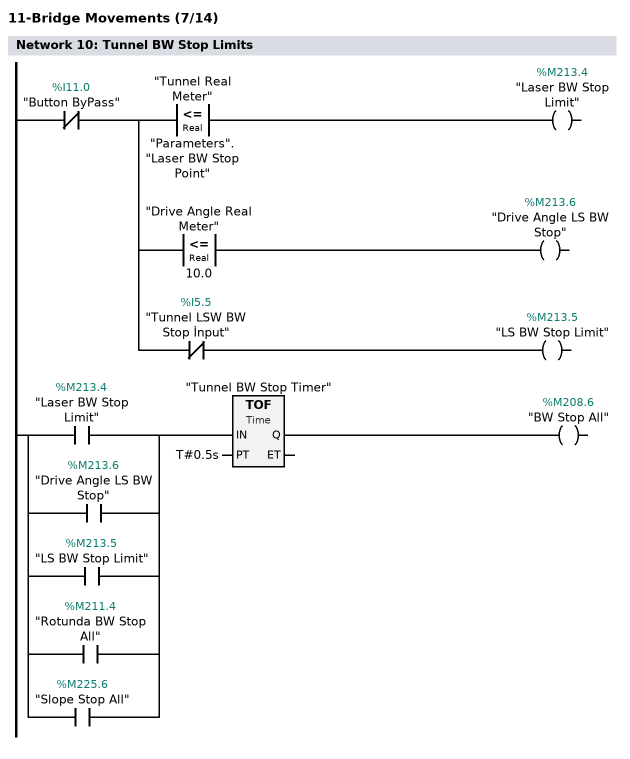
   RUNG wire#powerrail
      I_Contact( "Button ByPass" )
      wire#w1
      { S7_Templates := "SrcType := Real" } LE_Contact(in1 := "Tunnel Real Meter", in2 := "Parameters"."Laser BW Stop Point")
      Coil( "Laser BW Stop Limit" )
   END_RUNG
   RUNG wire#w1
      { S7_Templates := "SrcType := Real" } LE_Contact(in1 := "Drive Angle Real Meter", in2 := 10.0)
      Coil( "Drive Angle LS BW Stop" )
   END_RUNG
   RUNG wire#w1
      I_Contact( "Tunnel LSW BW Stop İnput" )
      Coil( "LS BW Stop Limit" )
   END_RUNG
   RUNG wire#powerrail
      Contact( "Laser BW Stop Limit" )
      wire#w2
      { S7_Templates := "time_type := Time" } "Tunnel BW Stop Timer".TOF(pt := T#0.5s, et =>)
      Coil( "BW Stop All" )
   END_RUNG
   RUNG wire#powerrail
      Contact( "Drive Angle LS BW Stop" )
   END_RUNG wire#w2
   RUNG wire#powerrail
      Contact( "LS BW Stop Limit" )
   END_RUNG wire#w2
   RUNG wire#powerrail
      Contact( "Rotunda BW Stop All" )
   END_RUNG wire#w2
   RUNG wire#powerrail
      Contact( "Slope Stop All" )
   END_RUNG wire#w2
   // the same network as SCL:
   "Laser BW Stop Limit" := NOT "Button ByPass" AND ("Tunnel Real Meter" <= "Parameters"."Laser BW Stop Point");
   "Drive Angle LS BW Stop" := NOT "Button ByPass" AND ("Drive Angle Real Meter" <= 10.0);
   "LS BW Stop Limit" := NOT "Button ByPass" AND NOT "Tunnel LSW BW Stop İnput";
   "Tunnel BW Stop Timer".TOF(IN := "Laser BW Stop Limit" OR "Drive Angle LS BW Stop" OR "LS BW Stop Limit" OR "Rotunda BW Stop All" OR "Slope Stop All",
                           PT := T#0.5s);
   "BW Stop All" := "Tunnel BW Stop Timer".Q;
END_REGION

REGION Network 11: Tunnel FW
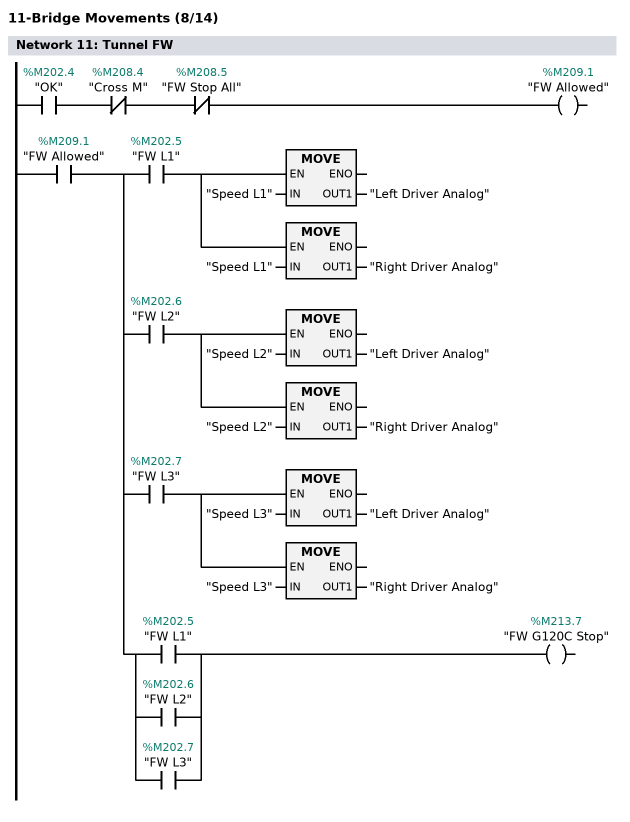
   RUNG wire#powerrail
      Contact( "OK" )
      I_Contact( "Cross M" )
      I_Contact( "FW Stop All" )
      Coil( "FW Allowed" )
   END_RUNG
   RUNG wire#powerrail
      Contact( "FW Allowed" )
      wire#w1
      Contact( "FW L1" )
      wire#w2
      Move(in := "Speed L1", out1 => "Left Driver Analog")
   END_RUNG
   RUNG wire#w2
      Move(in := "Speed L1", out1 => "Right Driver Analog")
   END_RUNG
   RUNG wire#w1
      Contact( "FW L2" )
      wire#w3
      Move(in := "Speed L2", out1 => "Left Driver Analog")
   END_RUNG
   RUNG wire#w3
      Move(in := "Speed L2", out1 => "Right Driver Analog")
   END_RUNG
   RUNG wire#w1
      Contact( "FW L3" )
      wire#w4
      Move(in := "Speed L3", out1 => "Left Driver Analog")
   END_RUNG
   RUNG wire#w4
      Move(in := "Speed L3", out1 => "Right Driver Analog")
   END_RUNG
   RUNG wire#w1
      Contact( "FW L1" )
      wire#w5
      Coil( "FW G120C Stop" )
   END_RUNG
   RUNG wire#w1
      Contact( "FW L2" )
   END_RUNG wire#w5
   RUNG wire#w1
      Contact( "FW L3" )
   END_RUNG wire#w5
   // the same network as SCL:
   "FW Allowed" := "OK" AND NOT "Cross M" AND NOT "FW Stop All";
   IF "FW Allowed" AND "FW L1" THEN
       "Left Driver Analog" := "Speed L1";
       "Right Driver Analog" := "Speed L1";
   END_IF;
   IF "FW Allowed" AND "FW L2" THEN
       "Left Driver Analog" := "Speed L2";
       "Right Driver Analog" := "Speed L2";
   END_IF;
   IF "FW Allowed" AND "FW L3" THEN
       "Left Driver Analog" := "Speed L3";
       "Right Driver Analog" := "Speed L3";
   END_IF;
   "FW G120C Stop" := "FW Allowed" AND ("FW L1" OR "FW L2" OR "FW L3");
END_REGION

REGION Network 12: Tunnel BW
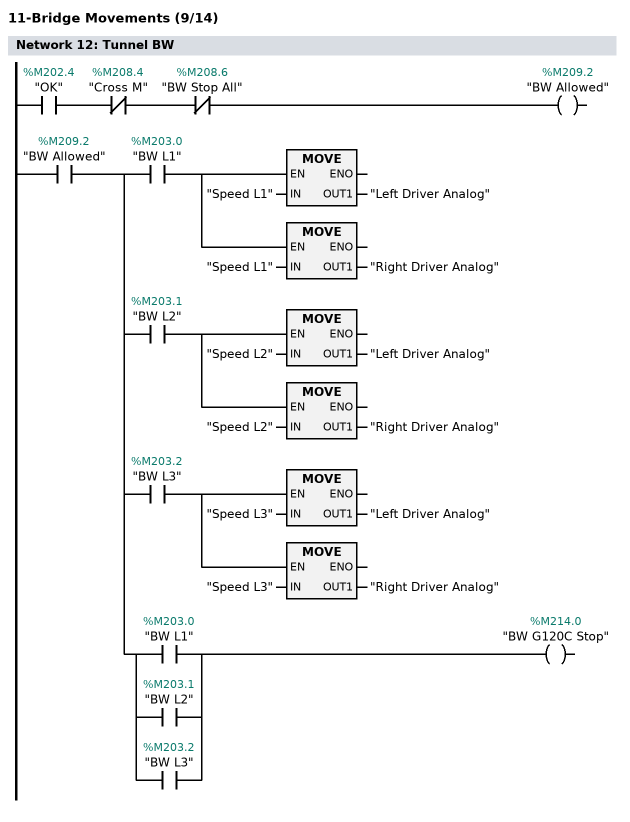
   RUNG wire#powerrail
      Contact( "OK" )
      I_Contact( "Cross M" )
      I_Contact( "BW Stop All" )
      Coil( "BW Allowed" )
   END_RUNG
   RUNG wire#powerrail
      Contact( "BW Allowed" )
      wire#w1
      Contact( "BW L1" )
      wire#w2
      Move(in := "Speed L1", out1 => "Left Driver Analog")
   END_RUNG
   RUNG wire#w2
      Move(in := "Speed L1", out1 => "Right Driver Analog")
   END_RUNG
   RUNG wire#w1
      Contact( "BW L2" )
      wire#w3
      Move(in := "Speed L2", out1 => "Left Driver Analog")
   END_RUNG
   RUNG wire#w3
      Move(in := "Speed L2", out1 => "Right Driver Analog")
   END_RUNG
   RUNG wire#w1
      Contact( "BW L3" )
      wire#w4
      Move(in := "Speed L3", out1 => "Left Driver Analog")
   END_RUNG
   RUNG wire#w4
      Move(in := "Speed L3", out1 => "Right Driver Analog")
   END_RUNG
   RUNG wire#w1
      Contact( "BW L1" )
      wire#w5
      Coil( "BW G120C Stop" )
   END_RUNG
   RUNG wire#w1
      Contact( "BW L2" )
   END_RUNG wire#w5
   RUNG wire#w1
      Contact( "BW L3" )
   END_RUNG wire#w5
   // the same network as SCL:
   "BW Allowed" := "OK" AND NOT "Cross M" AND NOT "BW Stop All";
   IF "BW Allowed" AND "BW L1" THEN
       "Left Driver Analog" := "Speed L1";
       "Right Driver Analog" := "Speed L1";
   END_IF;
   IF "BW Allowed" AND "BW L2" THEN
       "Left Driver Analog" := "Speed L2";
       "Right Driver Analog" := "Speed L2";
   END_IF;
   IF "BW Allowed" AND "BW L3" THEN
       "Left Driver Analog" := "Speed L3";
       "Right Driver Analog" := "Speed L3";
   END_IF;
   "BW G120C Stop" := "BW Allowed" AND ("BW L1" OR "BW L2" OR "BW L3");
END_REGION

REGION Network 13: Tunnel LFT
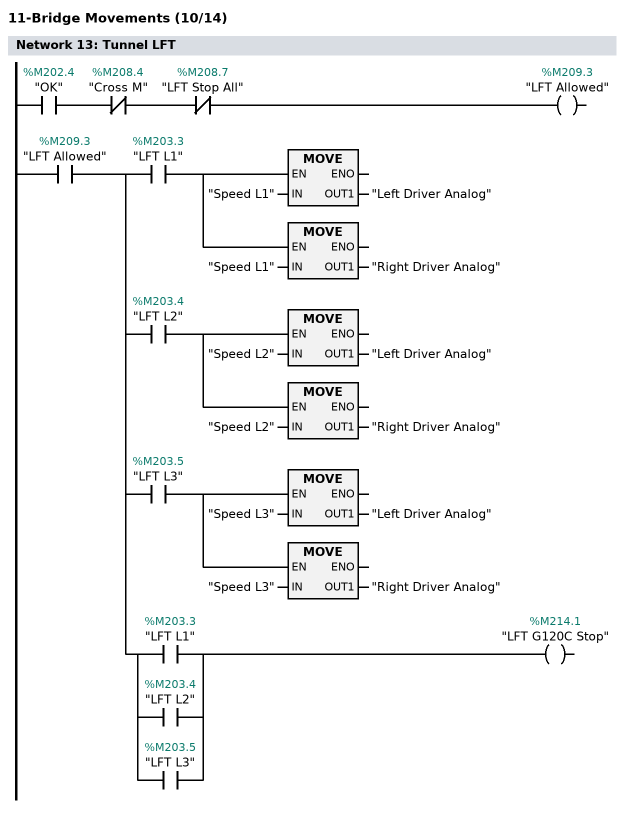
   RUNG wire#powerrail
      Contact( "OK" )
      I_Contact( "Cross M" )
      I_Contact( "LFT Stop All" )
      Coil( "LFT Allowed" )
   END_RUNG
   RUNG wire#powerrail
      Contact( "LFT Allowed" )
      wire#w1
      Contact( "LFT L1" )
      wire#w2
      Move(in := "Speed L1", out1 => "Left Driver Analog")
   END_RUNG
   RUNG wire#w2
      Move(in := "Speed L1", out1 => "Right Driver Analog")
   END_RUNG
   RUNG wire#w1
      Contact( "LFT L2" )
      wire#w3
      Move(in := "Speed L2", out1 => "Left Driver Analog")
   END_RUNG
   RUNG wire#w3
      Move(in := "Speed L2", out1 => "Right Driver Analog")
   END_RUNG
   RUNG wire#w1
      Contact( "LFT L3" )
      wire#w4
      Move(in := "Speed L3", out1 => "Left Driver Analog")
   END_RUNG
   RUNG wire#w4
      Move(in := "Speed L3", out1 => "Right Driver Analog")
   END_RUNG
   RUNG wire#w1
      Contact( "LFT L1" )
      wire#w5
      Coil( "LFT G120C Stop" )
   END_RUNG
   RUNG wire#w1
      Contact( "LFT L2" )
   END_RUNG wire#w5
   RUNG wire#w1
      Contact( "LFT L3" )
   END_RUNG wire#w5
   // the same network as SCL:
   "LFT Allowed" := "OK" AND NOT "Cross M" AND NOT "LFT Stop All";
   IF "LFT Allowed" AND "LFT L1" THEN
       "Left Driver Analog" := "Speed L1";
       "Right Driver Analog" := "Speed L1";
   END_IF;
   IF "LFT Allowed" AND "LFT L2" THEN
       "Left Driver Analog" := "Speed L2";
       "Right Driver Analog" := "Speed L2";
   END_IF;
   IF "LFT Allowed" AND "LFT L3" THEN
       "Left Driver Analog" := "Speed L3";
       "Right Driver Analog" := "Speed L3";
   END_IF;
   "LFT G120C Stop" := "LFT Allowed" AND ("LFT L1" OR "LFT L2" OR "LFT L3");
END_REGION

REGION Network 14: Tunnel RGHT
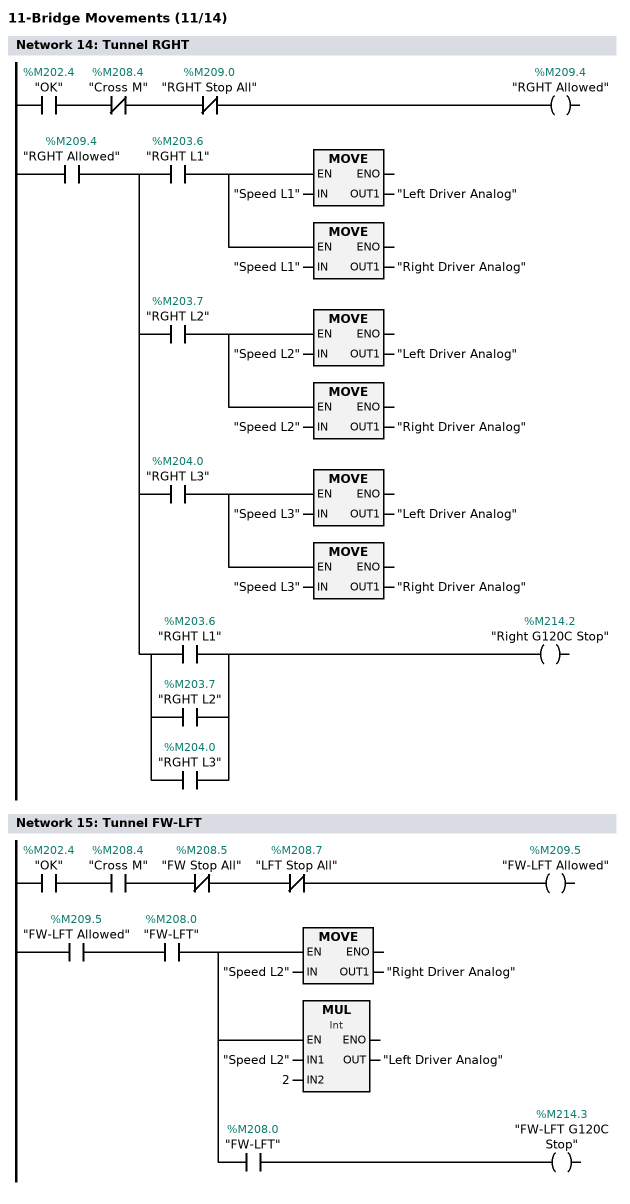
   RUNG wire#powerrail
      Contact( "OK" )
      I_Contact( "Cross M" )
      I_Contact( "RGHT Stop All" )
      Coil( "RGHT Allowed" )
   END_RUNG
   RUNG wire#powerrail
      Contact( "RGHT Allowed" )
      wire#w1
      Contact( "RGHT L1" )
      wire#w2
      Move(in := "Speed L1", out1 => "Left Driver Analog")
   END_RUNG
   RUNG wire#w2
      Move(in := "Speed L1", out1 => "Right Driver Analog")
   END_RUNG
   RUNG wire#w1
      Contact( "RGHT L2" )
      wire#w3
      Move(in := "Speed L2", out1 => "Left Driver Analog")
   END_RUNG
   RUNG wire#w3
      Move(in := "Speed L2", out1 => "Right Driver Analog")
   END_RUNG
   RUNG wire#w1
      Contact( "RGHT L3" )
      wire#w4
      Move(in := "Speed L3", out1 => "Left Driver Analog")
   END_RUNG
   RUNG wire#w4
      Move(in := "Speed L3", out1 => "Right Driver Analog")
   END_RUNG
   RUNG wire#w1
      Contact( "RGHT L1" )
      wire#w5
      Coil( "Right G120C Stop" )
   END_RUNG
   RUNG wire#w1
      Contact( "RGHT L2" )
   END_RUNG wire#w5
   RUNG wire#w1
      Contact( "RGHT L3" )
   END_RUNG wire#w5
   // the same network as SCL:
   "RGHT Allowed" := "OK" AND NOT "Cross M" AND NOT "RGHT Stop All";
   IF "RGHT Allowed" AND "RGHT L1" THEN
       "Left Driver Analog" := "Speed L1";
       "Right Driver Analog" := "Speed L1";
   END_IF;
   IF "RGHT Allowed" AND "RGHT L2" THEN
       "Left Driver Analog" := "Speed L2";
       "Right Driver Analog" := "Speed L2";
   END_IF;
   IF "RGHT Allowed" AND "RGHT L3" THEN
       "Left Driver Analog" := "Speed L3";
       "Right Driver Analog" := "Speed L3";
   END_IF;
   "Right G120C Stop" := "RGHT Allowed" AND ("RGHT L1" OR "RGHT L2" OR "RGHT L3");
END_REGION

REGION Network 15: Tunnel FW-LFT
   RUNG wire#powerrail
      Contact( "OK" )
      Contact( "Cross M" )
      I_Contact( "FW Stop All" )
      I_Contact( "LFT Stop All" )
      Coil( "FW-LFT Allowed" )
   END_RUNG
   RUNG wire#powerrail
      Contact( "FW-LFT Allowed" )
      Contact( "FW-LFT" )
      wire#w1
      Move(in := "Speed L2", out1 => "Right Driver Analog")
   END_RUNG
   RUNG wire#w1
      { S7_Templates := "SrcType := Int" } Mul(in1 := "Speed L2", in2 := 2, out => "Left Driver Analog")
   END_RUNG
   RUNG wire#w1
      Contact( "FW-LFT" )
      Coil( "FW-LFT G120C Stop" )
   END_RUNG
   // the same network as SCL:
   "FW-LFT Allowed" := "OK" AND "Cross M" AND NOT "FW Stop All" AND NOT "LFT Stop All";
   #_w1 := "FW-LFT Allowed" AND "FW-LFT";
   IF #_w1 THEN
       "Right Driver Analog" := "Speed L2";
       "Left Driver Analog" := "Speed L2" * 2;
   END_IF;
   "FW-LFT G120C Stop" := #_w1 AND "FW-LFT";
END_REGION

REGION Network 16: Tunnel FW-RGHT
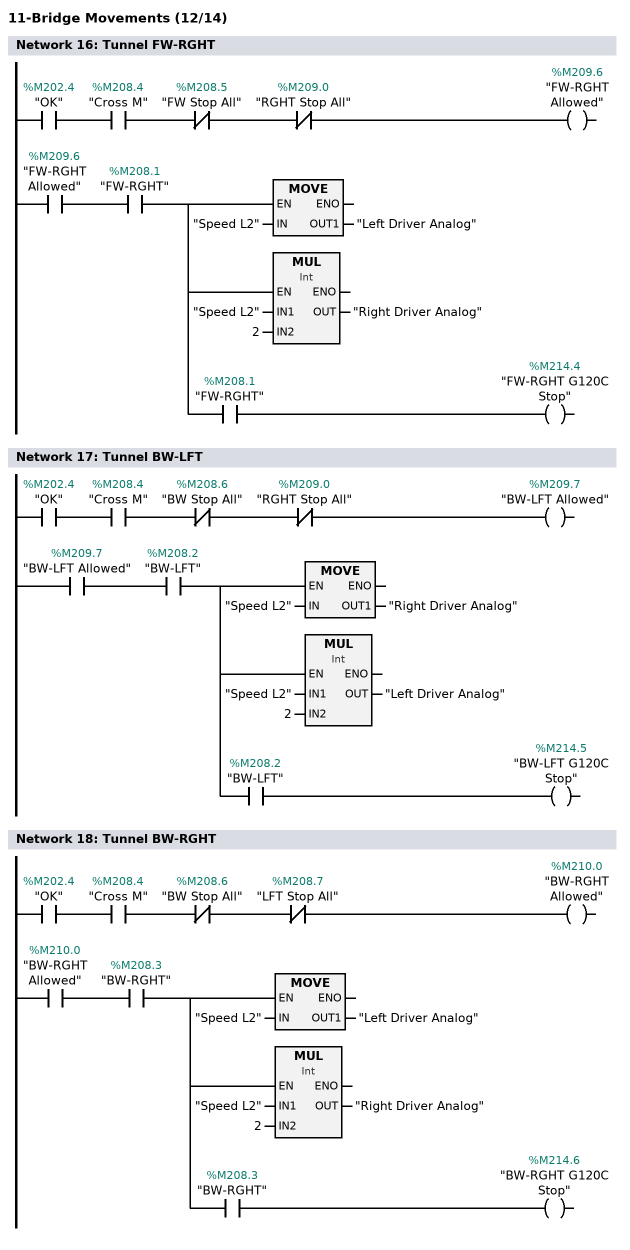
   RUNG wire#powerrail
      Contact( "OK" )
      Contact( "Cross M" )
      I_Contact( "FW Stop All" )
      I_Contact( "RGHT Stop All" )
      Coil( "FW-RGHT Allowed" )
   END_RUNG
   RUNG wire#powerrail
      Contact( "FW-RGHT Allowed" )
      Contact( "FW-RGHT" )
      wire#w1
      Move(in := "Speed L2", out1 => "Left Driver Analog")
   END_RUNG
   RUNG wire#w1
      { S7_Templates := "SrcType := Int" } Mul(in1 := "Speed L2", in2 := 2, out => "Right Driver Analog")
   END_RUNG
   RUNG wire#w1
      Contact( "FW-RGHT" )
      Coil( "FW-RGHT G120C Stop" )
   END_RUNG
   // the same network as SCL:
   "FW-RGHT Allowed" := "OK" AND "Cross M" AND NOT "FW Stop All" AND NOT "RGHT Stop All";
   #_w1 := "FW-RGHT Allowed" AND "FW-RGHT";
   IF #_w1 THEN
       "Left Driver Analog" := "Speed L2";
       "Right Driver Analog" := "Speed L2" * 2;
   END_IF;
   "FW-RGHT G120C Stop" := #_w1 AND "FW-RGHT";
END_REGION

REGION Network 17: Tunnel BW-LFT
   RUNG wire#powerrail
      Contact( "OK" )
      Contact( "Cross M" )
      I_Contact( "BW Stop All" )
      I_Contact( "RGHT Stop All" )
      Coil( "BW-LFT Allowed" )
   END_RUNG
   RUNG wire#powerrail
      Contact( "BW-LFT Allowed" )
      Contact( "BW-LFT" )
      wire#w1
      Move(in := "Speed L2", out1 => "Right Driver Analog")
   END_RUNG
   RUNG wire#w1
      { S7_Templates := "SrcType := Int" } Mul(in1 := "Speed L2", in2 := 2, out => "Left Driver Analog")
   END_RUNG
   RUNG wire#w1
      Contact( "BW-LFT" )
      Coil( "BW-LFT G120C Stop" )
   END_RUNG
   // the same network as SCL:
   "BW-LFT Allowed" := "OK" AND "Cross M" AND NOT "BW Stop All" AND NOT "RGHT Stop All";
   #_w1 := "BW-LFT Allowed" AND "BW-LFT";
   IF #_w1 THEN
       "Right Driver Analog" := "Speed L2";
       "Left Driver Analog" := "Speed L2" * 2;
   END_IF;
   "BW-LFT G120C Stop" := #_w1 AND "BW-LFT";
END_REGION

REGION Network 18: Tunnel BW-RGHT
   RUNG wire#powerrail
      Contact( "OK" )
      Contact( "Cross M" )
      I_Contact( "BW Stop All" )
      I_Contact( "LFT Stop All" )
      Coil( "BW-RGHT Allowed" )
   END_RUNG
   RUNG wire#powerrail
      Contact( "BW-RGHT Allowed" )
      Contact( "BW-RGHT" )
      wire#w1
      Move(in := "Speed L2", out1 => "Left Driver Analog")
   END_RUNG
   RUNG wire#w1
      { S7_Templates := "SrcType := Int" } Mul(in1 := "Speed L2", in2 := 2, out => "Right Driver Analog")
   END_RUNG
   RUNG wire#w1
      Contact( "BW-RGHT" )
      Coil( "BW-RGHT G120C Stop" )
   END_RUNG
   // the same network as SCL:
   "BW-RGHT Allowed" := "OK" AND "Cross M" AND NOT "BW Stop All" AND NOT "LFT Stop All";
   #_w1 := "BW-RGHT Allowed" AND "BW-RGHT";
   IF #_w1 THEN
       "Left Driver Analog" := "Speed L2";
       "Right Driver Analog" := "Speed L2" * 2;
   END_IF;
   "BW-RGHT G120C Stop" := #_w1 AND "BW-RGHT";
END_REGION

REGION Network 19: Drivers ON & Reversing !!!!
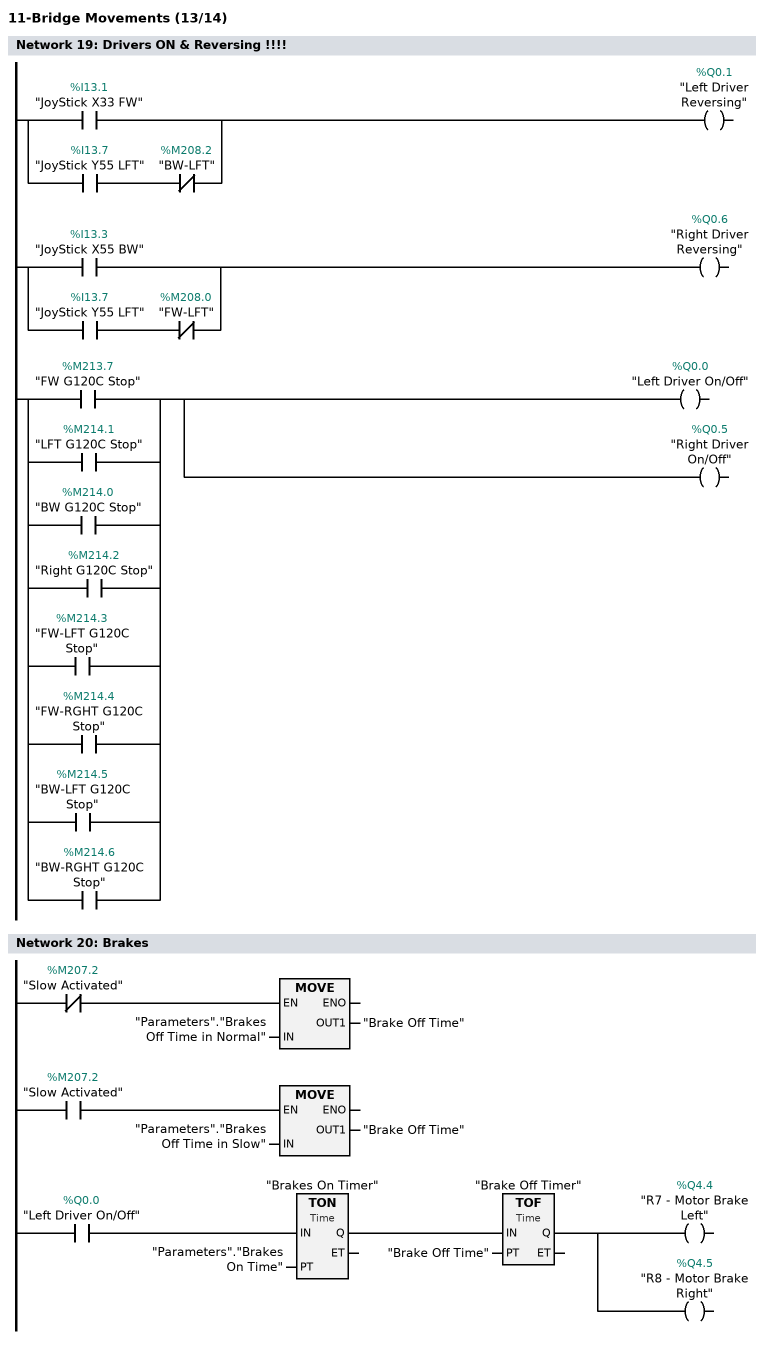
   RUNG wire#powerrail
      Contact( "JoyStick X33 FW" )
      wire#w1
      Coil( "Left Driver Reversing" )
   END_RUNG
   RUNG wire#powerrail
      Contact( "JoyStick Y55 LFT" )
      I_Contact( "BW-LFT" )
   END_RUNG wire#w1
   RUNG wire#powerrail
      Contact( "JoyStick X55 BW" )
      wire#w2
      Coil( "Right Driver Reversing" )
   END_RUNG
   RUNG wire#powerrail
      Contact( "JoyStick Y55 LFT" )
      I_Contact( "FW-LFT" )
   END_RUNG wire#w2
   RUNG wire#powerrail
      Contact( "FW G120C Stop" )
      wire#w3
      Coil( "Left Driver On/Off" )
   END_RUNG
   RUNG wire#powerrail
      Contact( "LFT G120C Stop" )
   END_RUNG wire#w3
   RUNG wire#powerrail
      Contact( "BW G120C Stop" )
   END_RUNG wire#w3
   RUNG wire#powerrail
      Contact( "Right G120C Stop" )
   END_RUNG wire#w3
   RUNG wire#powerrail
      Contact( "FW-LFT G120C Stop" )
   END_RUNG wire#w3
   RUNG wire#powerrail
      Contact( "FW-RGHT G120C Stop" )
   END_RUNG wire#w3
   RUNG wire#powerrail
      Contact( "BW-LFT G120C Stop" )
   END_RUNG wire#w3
   RUNG wire#powerrail
      Contact( "BW-RGHT G120C Stop" )
   END_RUNG wire#w3
   RUNG wire#w3
      Coil( "Right Driver On/Off" )
   END_RUNG
   // the same network as SCL:
   "Left Driver Reversing" := "JoyStick X33 FW" OR ("JoyStick Y55 LFT" AND NOT "BW-LFT");
   "Right Driver Reversing" := "JoyStick X55 BW" OR ("JoyStick Y55 LFT" AND NOT "FW-LFT");
   "Left Driver On/Off" := "FW G120C Stop" OR "LFT G120C Stop" OR "BW G120C Stop" OR "Right G120C Stop" OR "FW-LFT G120C Stop" OR "FW-RGHT G120C Stop" OR "BW-LFT G120C Stop" OR "BW-RGHT G120C Stop";
   "Right Driver On/Off" := "Left Driver On/Off";
END_REGION

REGION Network 20: Brakes
   RUNG wire#powerrail
      I_Contact( "Slow Activated" )
      Move(in := "Parameters"."Brakes Off Time in Normal", out1 => "Brake Off Time")
   END_RUNG
   RUNG wire#powerrail
      Contact( "Slow Activated" )
      Move(in := "Parameters"."Brakes Off Time in Slow", out1 => "Brake Off Time")
   END_RUNG
   RUNG wire#powerrail
      Contact( "Left Driver On/Off" )
      { S7_Templates := "time_type := Time" } "Brakes On Timer".TON(pt := "Parameters"."Brakes On Time", et =>)
      { S7_Templates := "time_type := Time" } "Brake Off Timer".TOF(pt := "Brake Off Time", et =>)
      wire#w1
      Coil( "R7 - Motor Brake Left" )
   END_RUNG
   RUNG wire#w1
      Coil( "R8 - Motor Brake Right" )
   END_RUNG
   // the same network as SCL:
   IF NOT "Slow Activated" THEN "Brake Off Time" := "Parameters"."Brakes Off Time in Normal"; END_IF;
   IF "Slow Activated" THEN "Brake Off Time" := "Parameters"."Brakes Off Time in Slow"; END_IF;
   "Brakes On Timer".TON(IN := "Left Driver On/Off", PT := "Parameters"."Brakes On Time");
   "Brake Off Timer".TOF(IN := "Brakes On Timer".Q, PT := "Brake Off Time");
   "R7 - Motor Brake Left" := "Brake Off Timer".Q;
   "R8 - Motor Brake Right" := "Brake Off Timer".Q;
END_REGION

REGION Network 21: SafetyEdge
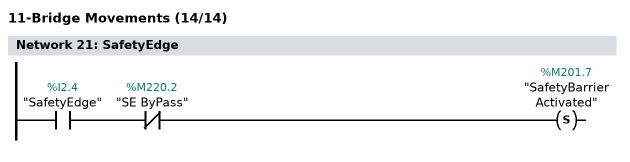
   RUNG wire#powerrail
      Contact( "SafetyEdge" )
      I_Contact( "SE ByPass" )
      S_Coil( "SafetyBarrier Activated" )
   END_RUNG
   // the same network as SCL:
   IF "SafetyEdge" AND NOT "SE ByPass" THEN "SafetyBarrier Activated" := TRUE; END_IF;
END_REGION
END_ORGANIZATION_BLOCK

ORGANIZATION_BLOCK "12-Drive Unit"   // OB131, LAD, ProgramCycle
TITLE = "Main Program Sweep (Cycle)"
{ S7_Optimized_Access := 'TRUE' }
VERSION : 0.1
// stored: AutoNumber true, IsIECCheckEnabled false, SetENOAutomatically false
   VAR_INPUT
      Initial_Call : Bool;   // Initial call of this OB
      Remanence : Bool;   // =True, if remanent data are available
   END_VAR
   VAR_TEMP
      "Drive Angle NomScale" : Real;
      "Drive Left Slow Point" : Real;
      tempory0 : Byte;
      tempory1 : Byte;
      "Drive Compare OK" : Bool;
      "Drive Right Slow Point" : Real;
   END_VAR
BEGIN

REGION Network 1: Drive Unit Angle Sensor
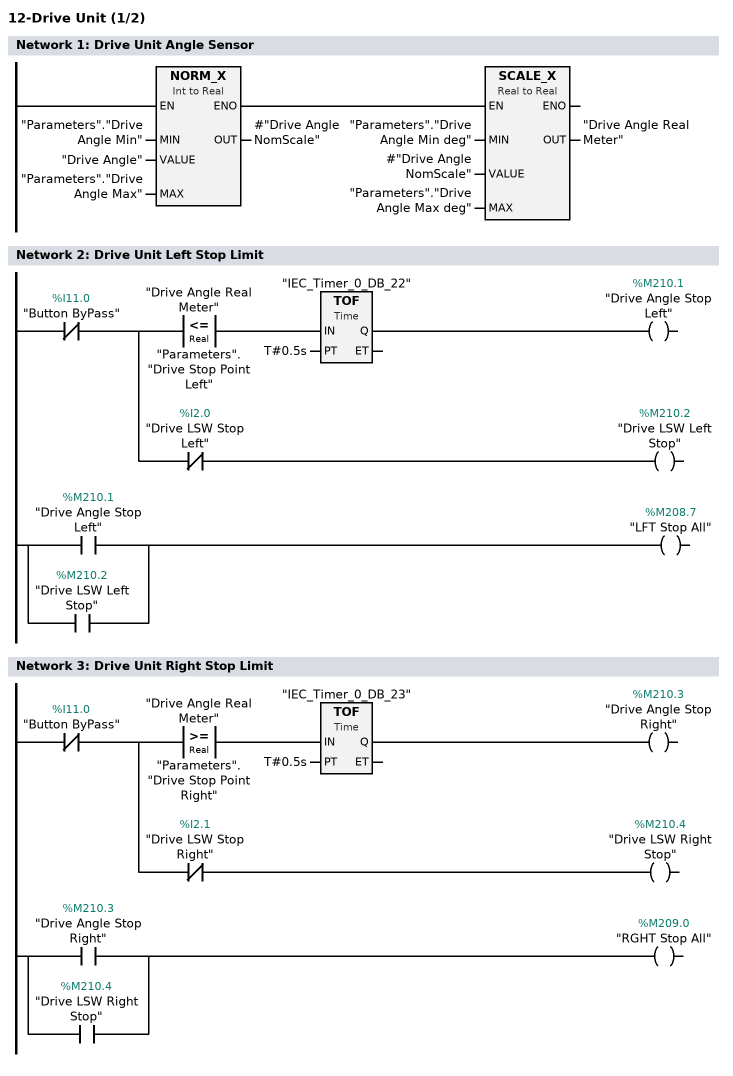
   RUNG wire#powerrail
      { S7_Templates := "[SrcType := Int, DestType := Real]" } Normalize(min := "Parameters"."Drive Angle Min", value := "Drive Angle", max := "Parameters"."Drive Angle Max", out => #"Drive Angle NomScale")
      { S7_Templates := "[SrcType := Real, DestType := Real]" } Scale(min := "Parameters"."Drive Angle Min deg", value := #"Drive Angle NomScale", max := "Parameters"."Drive Angle Max deg", out => "Drive Angle Real Meter")
   END_RUNG
   // the same network as SCL:
   #"Drive Angle NomScale" := NORM_X(MIN := "Parameters"."Drive Angle Min", VALUE := "Drive Angle", MAX := "Parameters"."Drive Angle Max");
   "Drive Angle Real Meter" := SCALE_X(MIN := "Parameters"."Drive Angle Min deg", VALUE := #"Drive Angle NomScale", MAX := "Parameters"."Drive Angle Max deg");
END_REGION

REGION Network 2: Drive Unit Left Stop Limit
   RUNG wire#powerrail
      I_Contact( "Button ByPass" )
      wire#w1
      { S7_Templates := "SrcType := Real" } LE_Contact(in1 := "Drive Angle Real Meter", in2 := "Parameters"."Drive Stop Point Left")
      { S7_Templates := "time_type := Time" } "IEC_Timer_0_DB_22".TOF(pt := T#0.5s, et =>)
      Coil( "Drive Angle Stop Left" )
   END_RUNG
   RUNG wire#w1
      I_Contact( "Drive LSW Stop Left" )
      Coil( "Drive LSW Left Stop" )
   END_RUNG
   RUNG wire#powerrail
      Contact( "Drive Angle Stop Left" )
      wire#w2
      Coil( "LFT Stop All" )
   END_RUNG
   RUNG wire#powerrail
      Contact( "Drive LSW Left Stop" )
   END_RUNG wire#w2
   // the same network as SCL:
   "IEC_Timer_0_DB_22".TOF(IN := NOT "Button ByPass" AND ("Drive Angle Real Meter" <= "Parameters"."Drive Stop Point Left"),
                           PT := T#0.5s);
   "Drive Angle Stop Left" := "IEC_Timer_0_DB_22".Q;
   "Drive LSW Left Stop" := NOT "Button ByPass" AND NOT "Drive LSW Stop Left";
   "LFT Stop All" := "Drive Angle Stop Left" OR "Drive LSW Left Stop";
END_REGION

REGION Network 3: Drive Unit Right Stop Limit
   RUNG wire#powerrail
      I_Contact( "Button ByPass" )
      wire#w1
      { S7_Templates := "SrcType := Real" } GE_Contact(in1 := "Drive Angle Real Meter", in2 := "Parameters"."Drive Stop Point Right")
      { S7_Templates := "time_type := Time" } "IEC_Timer_0_DB_23".TOF(pt := T#0.5s, et =>)
      Coil( "Drive Angle Stop Right" )
   END_RUNG
   RUNG wire#w1
      I_Contact( "Drive LSW Stop Right" )
      Coil( "Drive LSW Right Stop" )
   END_RUNG
   RUNG wire#powerrail
      Contact( "Drive Angle Stop Right" )
      wire#w2
      Coil( "RGHT Stop All" )
   END_RUNG
   RUNG wire#powerrail
      Contact( "Drive LSW Right Stop" )
   END_RUNG wire#w2
   // the same network as SCL:
   "IEC_Timer_0_DB_23".TOF(IN := NOT "Button ByPass" AND ("Drive Angle Real Meter" >= "Parameters"."Drive Stop Point Right"),
                           PT := T#0.5s);
   "Drive Angle Stop Right" := "IEC_Timer_0_DB_23".Q;
   "Drive LSW Right Stop" := NOT "Button ByPass" AND NOT "Drive LSW Stop Right";
   "RGHT Stop All" := "Drive Angle Stop Right" OR "Drive LSW Right Stop";
END_REGION

REGION Network 4: Drive Unit Slow Limits
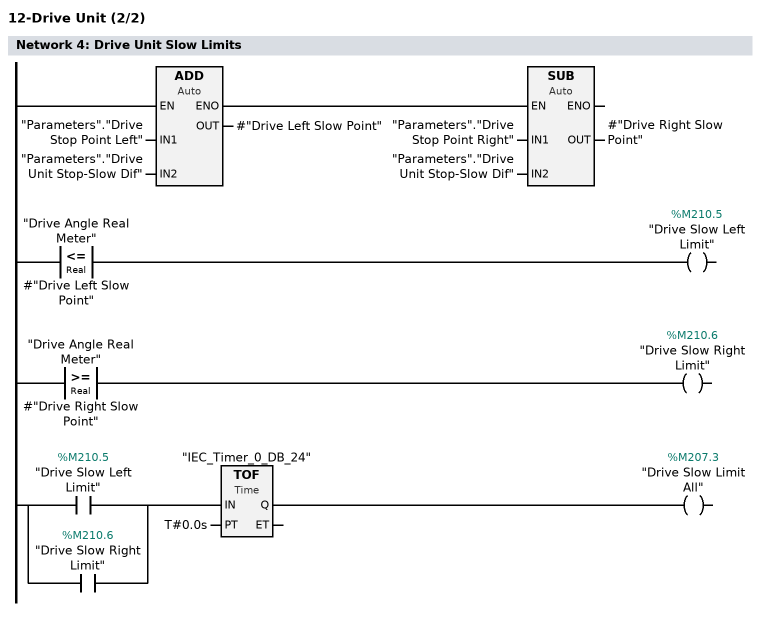
   RUNG wire#powerrail
      Add(in1 := "Parameters"."Drive Stop Point Left", in2 := "Parameters"."Drive Unit Stop-Slow Dif", out => #"Drive Left Slow Point")
      Sub(in1 := "Parameters"."Drive Stop Point Right", in2 := "Parameters"."Drive Unit Stop-Slow Dif", out => #"Drive Right Slow Point")
   END_RUNG
   RUNG wire#powerrail
      { S7_Templates := "SrcType := Real" } LE_Contact(in1 := "Drive Angle Real Meter", in2 := #"Drive Left Slow Point")
      Coil( "Drive Slow Left Limit" )
   END_RUNG
   RUNG wire#powerrail
      { S7_Templates := "SrcType := Real" } GE_Contact(in1 := "Drive Angle Real Meter", in2 := #"Drive Right Slow Point")
      Coil( "Drive Slow Right Limit" )
   END_RUNG
   RUNG wire#powerrail
      Contact( "Drive Slow Left Limit" )
      wire#w1
      { S7_Templates := "time_type := Time" } "IEC_Timer_0_DB_24".TOF(pt := T#0.0s, et =>)
      Coil( "Drive Slow Limit All" )
   END_RUNG
   RUNG wire#powerrail
      Contact( "Drive Slow Right Limit" )
   END_RUNG wire#w1
   // the same network as SCL:
   #"Drive Left Slow Point" := "Parameters"."Drive Stop Point Left" + "Parameters"."Drive Unit Stop-Slow Dif";
   #"Drive Right Slow Point" := "Parameters"."Drive Stop Point Right" - "Parameters"."Drive Unit Stop-Slow Dif";
   "Drive Slow Left Limit" := "Drive Angle Real Meter" <= #"Drive Left Slow Point";
   "Drive Slow Right Limit" := "Drive Angle Real Meter" >= #"Drive Right Slow Point";
   "IEC_Timer_0_DB_24".TOF(IN := "Drive Slow Left Limit" OR "Drive Slow Right Limit", PT := T#0.0s);
   "Drive Slow Limit All" := "IEC_Timer_0_DB_24".Q;
END_REGION
END_ORGANIZATION_BLOCK

ORGANIZATION_BLOCK "13-Laser Measure"   // OB132, LAD, ProgramCycle
TITLE = Laser / "Main Program Sweep (Cycle)"
{ S7_Optimized_Access := 'TRUE' }
VERSION : 0.1
// stored: AutoNumber true, IsIECCheckEnabled false, SetENOAutomatically false
   VAR_INPUT
      Initial_Call : Bool;   // Initial call of this OB
      Remanence : Bool;   // =True, if remanent data are available
   END_VAR
   VAR_TEMP
      "Laser NormScale" : Real;
   END_VAR
BEGIN

REGION Network 1: Laser
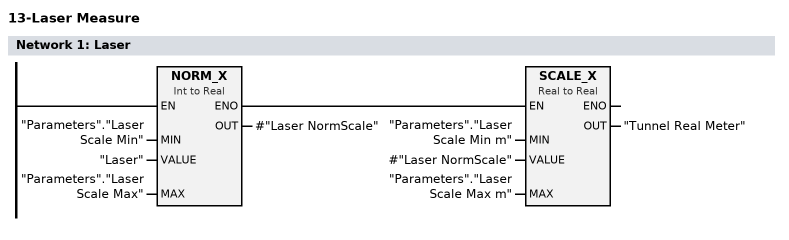
   RUNG wire#powerrail
      { S7_Templates := "[SrcType := Int, DestType := Real]" } Normalize(min := "Parameters"."Laser Scale Min", value := "Laser", max := "Parameters"."Laser Scale Max", out => #"Laser NormScale")
      { S7_Templates := "[SrcType := Real, DestType := Real]" } Scale(min := "Parameters"."Laser Scale Min m", value := #"Laser NormScale", max := "Parameters"."Laser Scale Max m", out => "Tunnel Real Meter")
   END_RUNG
   // the same network as SCL:
   #"Laser NormScale" := NORM_X(MIN := "Parameters"."Laser Scale Min", VALUE := "Laser", MAX := "Parameters"."Laser Scale Max");
   "Tunnel Real Meter" := SCALE_X(MIN := "Parameters"."Laser Scale Min m", VALUE := #"Laser NormScale", MAX := "Parameters"."Laser Scale Max m");
END_REGION
END_ORGANIZATION_BLOCK

ORGANIZATION_BLOCK "14-WireDraw"   // OB125, LAD, ProgramCycle
TITLE = "Main Program Sweep (Cycle)"
{ S7_Optimized_Access := 'TRUE' }
VERSION : 0.1
// stored: AutoNumber true, IsIECCheckEnabled false, SetENOAutomatically false
   VAR_INPUT
      Initial_Call : Bool;   // Initial call of this OB
      Remanence : Bool;   // =True, if remanent data are available
   END_VAR
   VAR_TEMP
      "Temp_1 (NormScale) Wire" : Real;
      "Temp_2 (NormScale) Inclanation" : Real;
      Temp_3 : Real;
      "Temp_4 (Radyan)" : Real;
      Temp_5 : Real;
   END_VAR
BEGIN

REGION Network 1: WireDraw Encoder _ Height Real
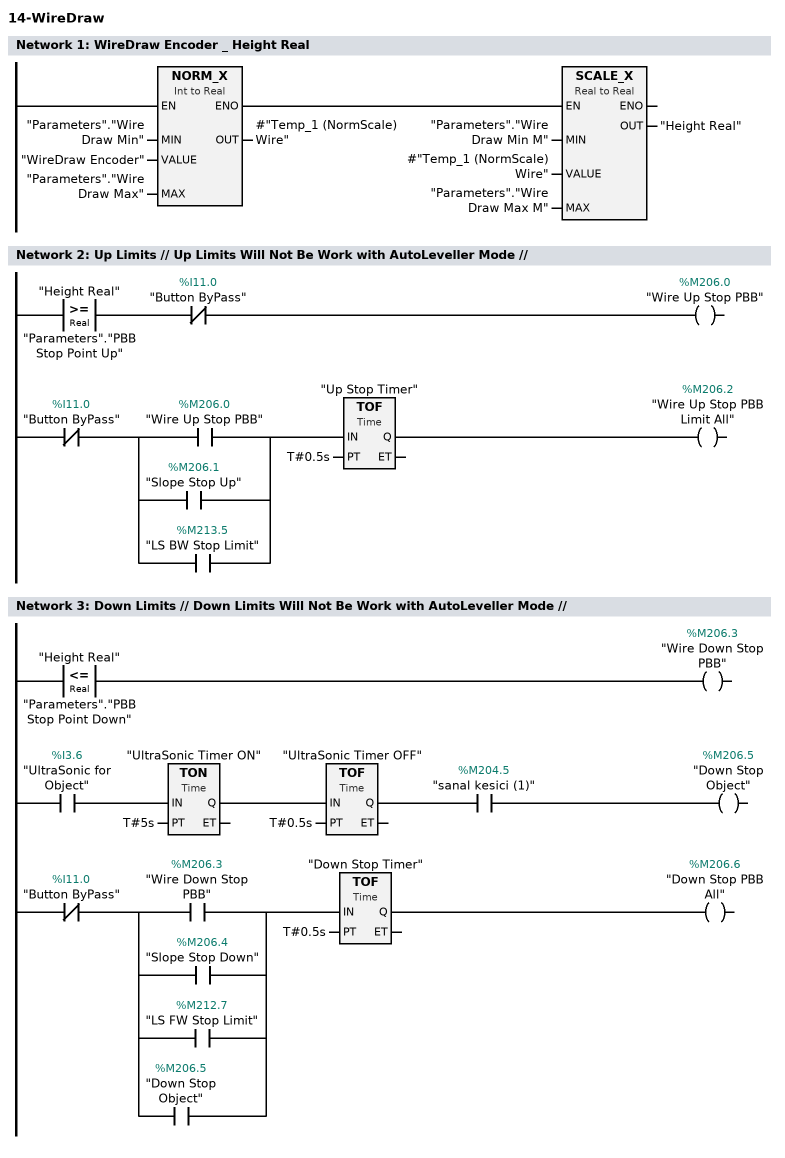
   RUNG wire#powerrail
      { S7_Templates := "[SrcType := Int, DestType := Real]" } Normalize(min := "Parameters"."Wire Draw Min", value := "WireDraw Encoder", max := "Parameters"."Wire Draw Max", out => #"Temp_1 (NormScale) Wire")
      { S7_Templates := "[SrcType := Real, DestType := Real]" } Scale(min := "Parameters"."Wire Draw Min M", value := #"Temp_1 (NormScale) Wire", max := "Parameters"."Wire Draw Max M", out => "Height Real")
   END_RUNG
   // the same network as SCL:
   #"Temp_1 (NormScale) Wire" := NORM_X(MIN := "Parameters"."Wire Draw Min", VALUE := "WireDraw Encoder", MAX := "Parameters"."Wire Draw Max");
   "Height Real" := SCALE_X(MIN := "Parameters"."Wire Draw Min M", VALUE := #"Temp_1 (NormScale) Wire", MAX := "Parameters"."Wire Draw Max M");
END_REGION

REGION Network 2: Up Limits // Up Limits Will Not Be Work with AutoLeveller Mode //
   RUNG wire#powerrail
      { S7_Templates := "SrcType := Real" } GE_Contact(in1 := "Height Real", in2 := "Parameters"."PBB Stop Point Up")
      I_Contact( "Button ByPass" )
      Coil( "Wire Up Stop PBB" )
   END_RUNG
   RUNG wire#powerrail
      I_Contact( "Button ByPass" )
      wire#w1
      Contact( "Wire Up Stop PBB" )
      wire#w2
      { S7_Templates := "time_type := Time" } "Up Stop Timer".TOF(pt := T#0.5s, et =>)
      Coil( "Wire Up Stop PBB Limit All" )
   END_RUNG
   RUNG wire#w1
      Contact( "Slope Stop Up" )
   END_RUNG wire#w2
   RUNG wire#w1
      Contact( "LS BW Stop Limit" )
   END_RUNG wire#w2
   // the same network as SCL:
   "Wire Up Stop PBB" := ("Height Real" >= "Parameters"."PBB Stop Point Up") AND NOT "Button ByPass";
   "Up Stop Timer".TOF(IN := NOT "Button ByPass" AND ("Wire Up Stop PBB" OR "Slope Stop Up" OR "LS BW Stop Limit"),
                       PT := T#0.5s);
   "Wire Up Stop PBB Limit All" := "Up Stop Timer".Q;
END_REGION

REGION Network 3: Down Limits // Down Limits Will Not Be Work with AutoLeveller Mode //
   RUNG wire#powerrail
      { S7_Templates := "SrcType := Real" } LE_Contact(in1 := "Height Real", in2 := "Parameters"."PBB Stop Point Down")
      Coil( "Wire Down Stop PBB" )
   END_RUNG
   RUNG wire#powerrail
      Contact( "UltraSonic for Object" )
      { S7_Templates := "time_type := Time" } "UltraSonic Timer ON".TON(pt := T#5s, et =>)
      { S7_Templates := "time_type := Time" } "UltraSonic Timer OFF".TOF(pt := T#0.5s, et =>)
      Contact( "sanal kesici (1)" )
      Coil( "Down Stop Object" )
   END_RUNG
   RUNG wire#powerrail
      I_Contact( "Button ByPass" )
      wire#w1
      Contact( "Wire Down Stop PBB" )
      wire#w2
      { S7_Templates := "time_type := Time" } "Down Stop Timer".TOF(pt := T#0.5s, et =>)
      Coil( "Down Stop PBB All" )
   END_RUNG
   RUNG wire#w1
      Contact( "Slope Stop Down" )
   END_RUNG wire#w2
   RUNG wire#w1
      Contact( "LS FW Stop Limit" )
   END_RUNG wire#w2
   RUNG wire#w1
      Contact( "Down Stop Object" )
   END_RUNG wire#w2
   // the same network as SCL:
   "Wire Down Stop PBB" := "Height Real" <= "Parameters"."PBB Stop Point Down";
   "UltraSonic Timer ON".TON(IN := "UltraSonic for Object", PT := T#5s);
   "UltraSonic Timer OFF".TOF(IN := "UltraSonic Timer ON".Q, PT := T#0.5s);
   "Down Stop Object" := "UltraSonic Timer OFF".Q AND "sanal kesici (1)";
   "Down Stop Timer".TOF(IN := NOT "Button ByPass" AND ("Wire Down Stop PBB" OR "Slope Stop Down" OR "LS FW Stop Limit" OR "Down Stop Object"),
                         PT := T#0.5s);
   "Down Stop PBB All" := "Down Stop Timer".Q;
END_REGION
END_ORGANIZATION_BLOCK

ORGANIZATION_BLOCK "15-Slope"   // OB128, LAD, ProgramCycle
TITLE = "Main Program Sweep (Cycle)"
{ S7_Optimized_Access := 'TRUE' }
VERSION : 0.1
// stored: AutoNumber true, IsIECCheckEnabled false, SetENOAutomatically false
   VAR_INPUT
      Initial_Call : Bool;   // Initial call of this OB
      Remanence : Bool;   // =True, if remanent data are available
   END_VAR
   VAR_TEMP
      "Temp_1 (NormScale) Wire" : Real;
      "Temp_2 (NormScale) Inclanation" : Real;
      Temp_3 : Real;
      "Temp_4 (Radyan)" : Real;
      Temp_5 : Real;
      "Temp-6 AnimasyonNorm" : Real;
   END_VAR
BEGIN

REGION Network 1: Slope Angle
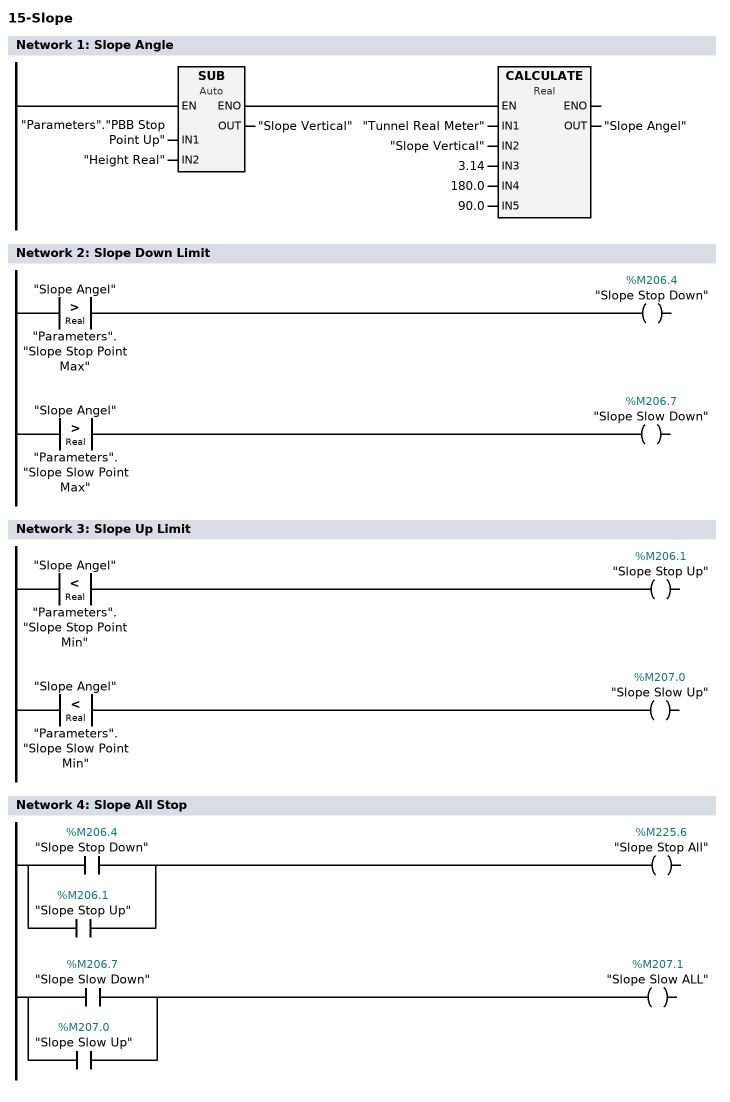
   RUNG wire#powerrail
      Sub(in1 := "Parameters"."PBB Stop Point Up", in2 := "Height Real", out => "Slope Vertical")
      { S7_Templates := "SrcType := Real"; S7_Expression := "IN5 -((ACOS(IN2 / IN1) *IN4) / IN3)" } Calculate(in1 := "Tunnel Real Meter", in2 := "Slope Vertical", in3 := 3.14, in4 := 180.0, in5 := 90.0, out => "Slope Angel")
   END_RUNG
   // the same network as SCL:
   "Slope Vertical" := "Parameters"."PBB Stop Point Up" - "Height Real";
   "Slope Angel" := 90.0 -((ACOS("Slope Vertical" / "Tunnel Real Meter") *180.0) / 3.14);
END_REGION

REGION Network 2: Slope Down Limit
   RUNG wire#powerrail
      { S7_Templates := "SrcType := Real" } GT_Contact(in1 := "Slope Angel", in2 := "Parameters"."Slope Stop Point Max")
      Coil( "Slope Stop Down" )
   END_RUNG
   RUNG wire#powerrail
      { S7_Templates := "SrcType := Real" } GT_Contact(in1 := "Slope Angel", in2 := "Parameters"."Slope Slow Point Max")
      Coil( "Slope Slow Down" )
   END_RUNG
   // the same network as SCL:
   "Slope Stop Down" := "Slope Angel" > "Parameters"."Slope Stop Point Max";
   "Slope Slow Down" := "Slope Angel" > "Parameters"."Slope Slow Point Max";
END_REGION

REGION Network 3: Slope Up Limit
   RUNG wire#powerrail
      { S7_Templates := "SrcType := Real" } LT_Contact(in1 := "Slope Angel", in2 := "Parameters"."Slope Stop Point Min")
      Coil( "Slope Stop Up" )
   END_RUNG
   RUNG wire#powerrail
      { S7_Templates := "SrcType := Real" } LT_Contact(in1 := "Slope Angel", in2 := "Parameters"."Slope Slow Point Min")
      Coil( "Slope Slow Up" )
   END_RUNG
   // the same network as SCL:
   "Slope Stop Up" := "Slope Angel" < "Parameters"."Slope Stop Point Min";
   "Slope Slow Up" := "Slope Angel" < "Parameters"."Slope Slow Point Min";
END_REGION

REGION Network 4: Slope All Stop
   RUNG wire#powerrail
      Contact( "Slope Stop Down" )
      wire#w1
      Coil( "Slope Stop All" )
   END_RUNG
   RUNG wire#powerrail
      Contact( "Slope Stop Up" )
   END_RUNG wire#w1
   RUNG wire#powerrail
      Contact( "Slope Slow Down" )
      wire#w2
      Coil( "Slope Slow ALL" )
   END_RUNG
   RUNG wire#powerrail
      Contact( "Slope Slow Up" )
   END_RUNG wire#w2
   // the same network as SCL:
   "Slope Stop All" := "Slope Stop Down" OR "Slope Stop Up";
   "Slope Slow ALL" := "Slope Slow Down" OR "Slope Slow Up";
END_REGION
END_ORGANIZATION_BLOCK

ORGANIZATION_BLOCK "16-Rotunda"   // OB130, LAD, ProgramCycle
TITLE = Rotunda / "Main Program Sweep (Cycle)"
{ S7_Optimized_Access := 'TRUE' }
VERSION : 0.1
// stored: AutoNumber true, IsIECCheckEnabled false, SetENOAutomatically false
   VAR_INPUT
      Initial_Call : Bool;   // Initial call of this OB
      Remanence : Bool;   // =True, if remanent data are available
   END_VAR
   VAR_TEMP
      "Angle Rotunda NormScale" : Real;
   END_VAR
   VAR_TEMP   // added for the SCL form of the ladder/FBD networks
      _w1 : Bool;
      _w2 : Bool;
   END_VAR
BEGIN

REGION Network 1: Rotunda Angle Sensor
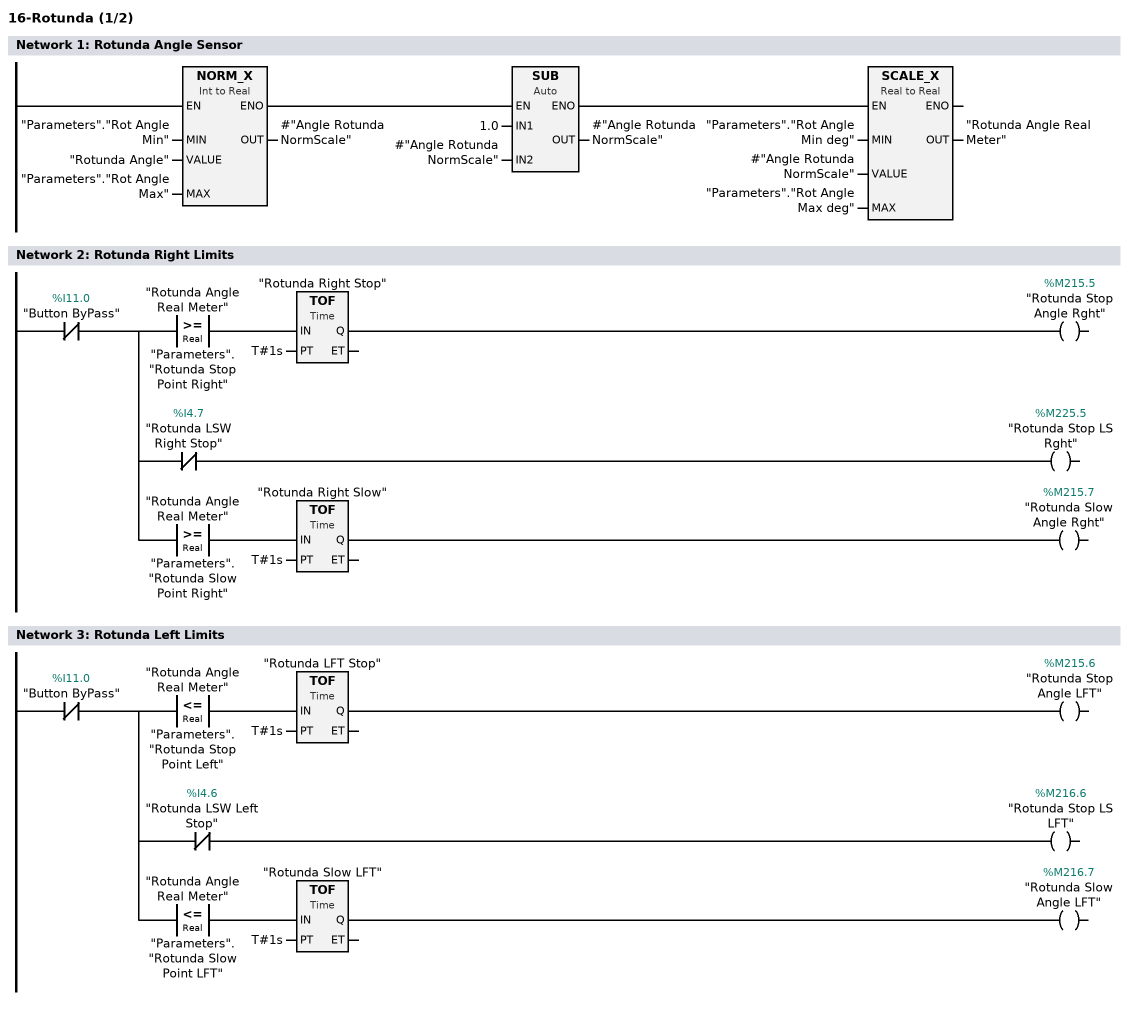
   RUNG wire#powerrail
      { S7_Templates := "[SrcType := Int, DestType := Real]" } Normalize(min := "Parameters"."Rot Angle Min", value := "Rotunda Angle", max := "Parameters"."Rot Angle Max", out => #"Angle Rotunda NormScale")
      Sub(in1 := 1.0, in2 := #"Angle Rotunda NormScale", out => #"Angle Rotunda NormScale")
      { S7_Templates := "[SrcType := Real, DestType := Real]" } Scale(min := "Parameters"."Rot Angle Min deg", value := #"Angle Rotunda NormScale", max := "Parameters"."Rot Angle Max deg", out => "Rotunda Angle Real Meter")
   END_RUNG
   // the same network as SCL:
   #"Angle Rotunda NormScale" := NORM_X(MIN := "Parameters"."Rot Angle Min", VALUE := "Rotunda Angle", MAX := "Parameters"."Rot Angle Max");
   #"Angle Rotunda NormScale" := 1.0 - #"Angle Rotunda NormScale";
   "Rotunda Angle Real Meter" := SCALE_X(MIN := "Parameters"."Rot Angle Min deg", VALUE := #"Angle Rotunda NormScale", MAX := "Parameters"."Rot Angle Max deg");
END_REGION

REGION Network 2: Rotunda Right Limits
   RUNG wire#powerrail
      I_Contact( "Button ByPass" )
      wire#w1
      { S7_Templates := "SrcType := Real" } GE_Contact(in1 := "Rotunda Angle Real Meter", in2 := "Parameters"."Rotunda Stop Point Right")
      { S7_Templates := "time_type := Time" } "Rotunda Right Stop".TOF(pt := T#1s, et =>)
      Coil( "Rotunda Stop Angle Rght" )
   END_RUNG
   RUNG wire#w1
      I_Contact( "Rotunda LSW Right Stop" )
      Coil( "Rotunda Stop LS Rght" )
   END_RUNG
   RUNG wire#w1
      { S7_Templates := "SrcType := Real" } GE_Contact(in1 := "Rotunda Angle Real Meter", in2 := "Parameters"."Rotunda Slow Point Right")
      { S7_Templates := "time_type := Time" } "Rotunda Right Slow".TOF(pt := T#1s, et =>)
      Coil( "Rotunda Slow Angle Rght" )
   END_RUNG
   // the same network as SCL:
   "Rotunda Right Stop".TOF(IN := NOT "Button ByPass" AND ("Rotunda Angle Real Meter" >= "Parameters"."Rotunda Stop Point Right"),
                           PT := T#1s);
   "Rotunda Stop Angle Rght" := "Rotunda Right Stop".Q;
   "Rotunda Stop LS Rght" := NOT "Button ByPass" AND NOT "Rotunda LSW Right Stop";
   "Rotunda Right Slow".TOF(IN := NOT "Button ByPass" AND ("Rotunda Angle Real Meter" >= "Parameters"."Rotunda Slow Point Right"),
                           PT := T#1s);
   "Rotunda Slow Angle Rght" := "Rotunda Right Slow".Q;
END_REGION

REGION Network 3: Rotunda Left Limits
   RUNG wire#powerrail
      I_Contact( "Button ByPass" )
      wire#w1
      { S7_Templates := "SrcType := Real" } LE_Contact(in1 := "Rotunda Angle Real Meter", in2 := "Parameters"."Rotunda Stop Point Left")
      { S7_Templates := "time_type := Time" } "Rotunda LFT Stop".TOF(pt := T#1s, et =>)
      Coil( "Rotunda Stop Angle LFT" )
   END_RUNG
   RUNG wire#w1
      I_Contact( "Rotunda LSW Left Stop" )
      Coil( "Rotunda Stop LS LFT" )
   END_RUNG
   RUNG wire#w1
      { S7_Templates := "SrcType := Real" } LE_Contact(in1 := "Rotunda Angle Real Meter", in2 := "Parameters"."Rotunda Slow Point LFT")
      { S7_Templates := "time_type := Time" } "Rotunda Slow LFT".TOF(pt := T#1s, et =>)
      Coil( "Rotunda Slow Angle LFT" )
   END_RUNG
   // the same network as SCL:
   "Rotunda LFT Stop".TOF(IN := NOT "Button ByPass" AND ("Rotunda Angle Real Meter" <= "Parameters"."Rotunda Stop Point Left"),
                          PT := T#1s);
   "Rotunda Stop Angle LFT" := "Rotunda LFT Stop".Q;
   "Rotunda Stop LS LFT" := NOT "Button ByPass" AND NOT "Rotunda LSW Left Stop";
   "Rotunda Slow LFT".TOF(IN := NOT "Button ByPass" AND ("Rotunda Angle Real Meter" <= "Parameters"."Rotunda Slow Point LFT"),
                          PT := T#1s);
   "Rotunda Slow Angle LFT" := "Rotunda Slow LFT".Q;
END_REGION

REGION Network 4: Rotunda Stop-Slow Limits
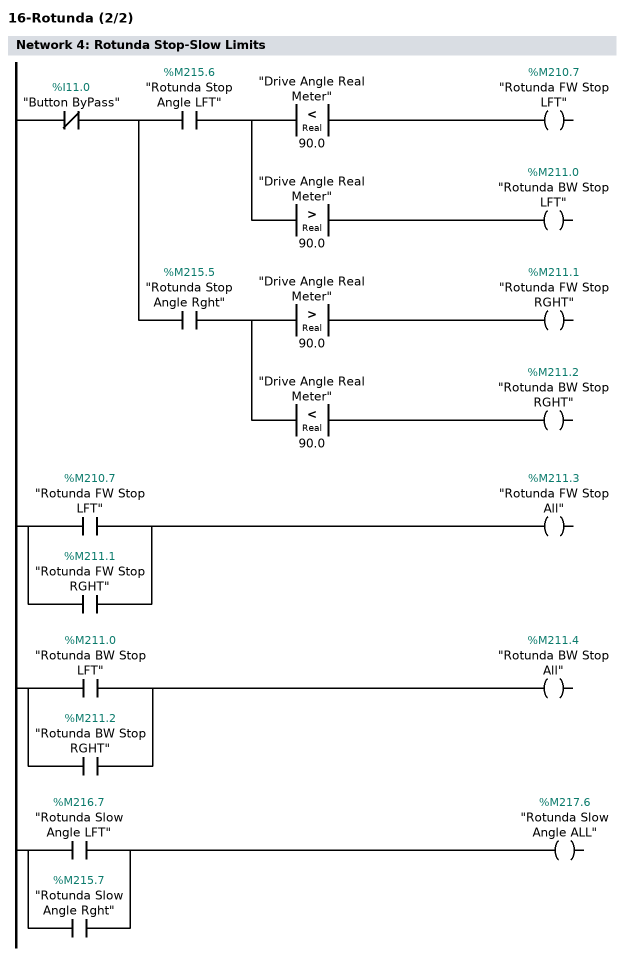
   RUNG wire#powerrail
      I_Contact( "Button ByPass" )
      wire#w1
      Contact( "Rotunda Stop Angle LFT" )
      wire#w2
      { S7_Templates := "SrcType := Real" } LT_Contact(in1 := "Drive Angle Real Meter", in2 := 90.0)
      Coil( "Rotunda FW Stop LFT" )
   END_RUNG
   RUNG wire#w2
      { S7_Templates := "SrcType := Real" } GT_Contact(in1 := "Drive Angle Real Meter", in2 := 90.0)
      Coil( "Rotunda BW Stop LFT" )
   END_RUNG
   RUNG wire#w1
      Contact( "Rotunda Stop Angle Rght" )
      wire#w3
      { S7_Templates := "SrcType := Real" } GT_Contact(in1 := "Drive Angle Real Meter", in2 := 90.0)
      Coil( "Rotunda FW Stop RGHT" )
   END_RUNG
   RUNG wire#w3
      { S7_Templates := "SrcType := Real" } LT_Contact(in1 := "Drive Angle Real Meter", in2 := 90.0)
      Coil( "Rotunda BW Stop RGHT" )
   END_RUNG
   RUNG wire#powerrail
      Contact( "Rotunda FW Stop LFT" )
      wire#w4
      Coil( "Rotunda FW Stop All" )
   END_RUNG
   RUNG wire#powerrail
      Contact( "Rotunda FW Stop RGHT" )
   END_RUNG wire#w4
   RUNG wire#powerrail
      Contact( "Rotunda BW Stop LFT" )
      wire#w5
      Coil( "Rotunda BW Stop All" )
   END_RUNG
   RUNG wire#powerrail
      Contact( "Rotunda BW Stop RGHT" )
   END_RUNG wire#w5
   RUNG wire#powerrail
      Contact( "Rotunda Slow Angle LFT" )
      wire#w6
      Coil( "Rotunda Slow Angle ALL" )
   END_RUNG
   RUNG wire#powerrail
      Contact( "Rotunda Slow Angle Rght" )
   END_RUNG wire#w6
   // the same network as SCL:
   #_w1 := NOT "Button ByPass" AND "Rotunda Stop Angle LFT";
   "Rotunda FW Stop LFT" := #_w1 AND ("Drive Angle Real Meter" < 90.0);
   "Rotunda BW Stop LFT" := #_w1 AND ("Drive Angle Real Meter" > 90.0);
   #_w2 := NOT "Button ByPass" AND "Rotunda Stop Angle Rght";
   "Rotunda FW Stop RGHT" := #_w2 AND ("Drive Angle Real Meter" > 90.0);
   "Rotunda BW Stop RGHT" := #_w2 AND ("Drive Angle Real Meter" < 90.0);
   "Rotunda FW Stop All" := "Rotunda FW Stop LFT" OR "Rotunda FW Stop RGHT";
   "Rotunda BW Stop All" := "Rotunda BW Stop LFT" OR "Rotunda BW Stop RGHT";
   "Rotunda Slow Angle ALL" := "Rotunda Slow Angle LFT" OR "Rotunda Slow Angle Rght";
END_REGION
END_ORGANIZATION_BLOCK

ORGANIZATION_BLOCK "17-Cabin Movement"   // OB124, LAD, ProgramCycle
TITLE = "Main Program Sweep (Cycle)"
{ S7_Optimized_Access := 'TRUE' }
VERSION : 0.1
// stored: AutoNumber true, IsIECCheckEnabled false, SetENOAutomatically false
   VAR_INPUT
      Initial_Call : Bool;   // Initial call of this OB
      Remanence : Bool;   // =True, if remanent data are available
   END_VAR
   VAR_TEMP
      "Cab Angle NormScale" : Real;
   END_VAR
BEGIN

REGION Network 1: Cab Movement
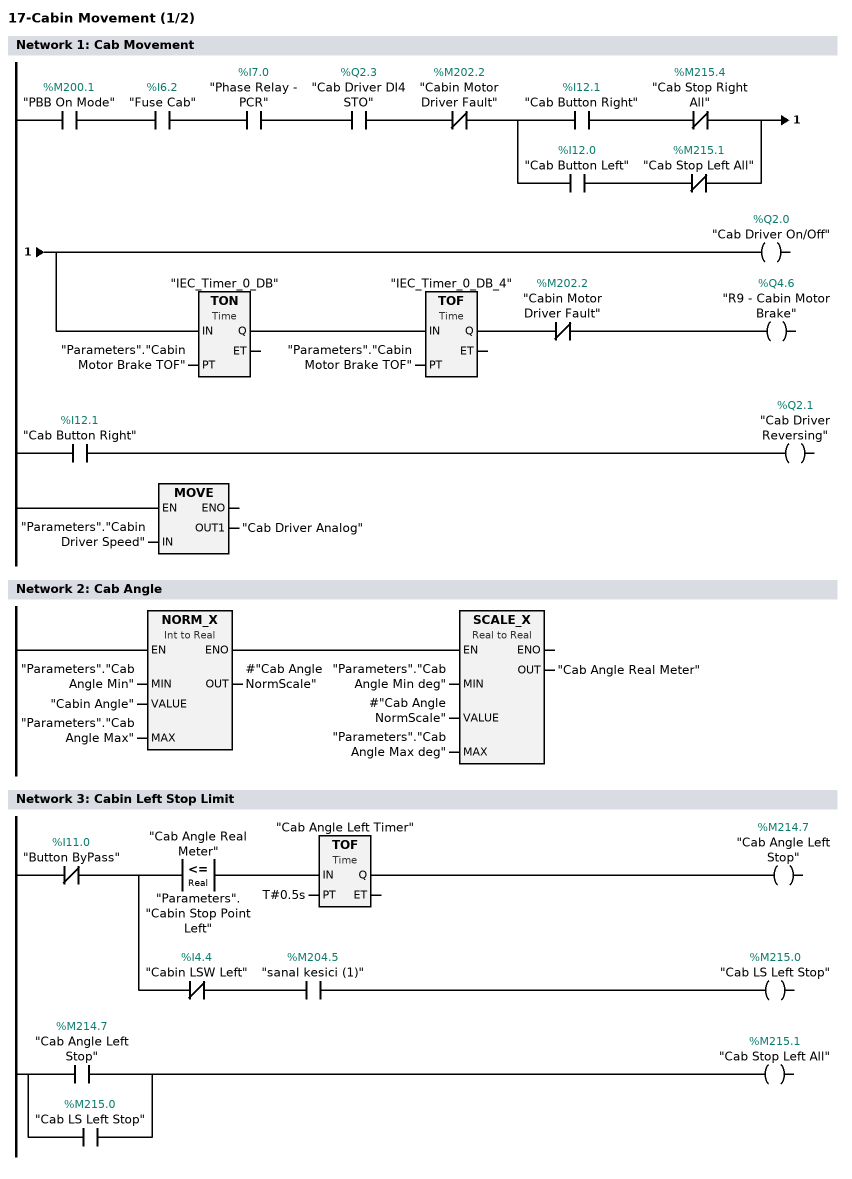
   RUNG wire#powerrail
      Contact( "PBB On Mode" )
      Contact( "Fuse Cab" )
      Contact( "Phase Relay - PCR" )
      Contact( "Cab Driver DI4 STO" )
      I_Contact( "Cabin Motor Driver Fault" )
      wire#w1
      Contact( "Cab Button Right" )
      I_Contact( "Cab Stop Right All" )
      wire#w2
      Coil( "Cab Driver On/Off" )
   END_RUNG
   RUNG wire#w1
      Contact( "Cab Button Left" )
      I_Contact( "Cab Stop Left All" )
   END_RUNG wire#w2
   RUNG wire#w2
      { S7_Templates := "time_type := Time" } "IEC_Timer_0_DB".TON(pt := "Parameters"."Cabin Motor Brake TOF", et =>)
      { S7_Templates := "time_type := Time" } "IEC_Timer_0_DB_4".TOF(pt := "Parameters"."Cabin Motor Brake TOF", et =>)
      I_Contact( "Cabin Motor Driver Fault" )
      Coil( "R9 - Cabin Motor Brake" )
   END_RUNG
   RUNG wire#powerrail
      Contact( "Cab Button Right" )
      Coil( "Cab Driver Reversing" )
   END_RUNG
   RUNG wire#powerrail
      Move(in := "Parameters"."Cabin Driver Speed", out1 => "Cab Driver Analog")
   END_RUNG
   // the same network as SCL:
   "Cab Driver On/Off" := "PBB On Mode" AND "Fuse Cab" AND "Phase Relay - PCR" AND "Cab Driver DI4 STO" AND NOT "Cabin Motor Driver Fault" AND (("Cab Button Right" AND NOT "Cab Stop Right All") OR ("Cab Button Left" AND NOT "Cab Stop Left All"));
   "IEC_Timer_0_DB".TON(IN := "Cab Driver On/Off", PT := "Parameters"."Cabin Motor Brake TOF");
   "IEC_Timer_0_DB_4".TOF(IN := "IEC_Timer_0_DB".Q, PT := "Parameters"."Cabin Motor Brake TOF");
   "R9 - Cabin Motor Brake" := "IEC_Timer_0_DB_4".Q AND NOT "Cabin Motor Driver Fault";
   "Cab Driver Reversing" := "Cab Button Right";
   "Cab Driver Analog" := "Parameters"."Cabin Driver Speed";
END_REGION

REGION Network 2: Cab Angle
   RUNG wire#powerrail
      { S7_Templates := "[SrcType := Int, DestType := Real]" } Normalize(min := "Parameters"."Cab Angle Min", value := "Cabin Angle", max := "Parameters"."Cab Angle Max", out => #"Cab Angle NormScale")
      { S7_Templates := "[SrcType := Real, DestType := Real]" } Scale(min := "Parameters"."Cab Angle Min deg", value := #"Cab Angle NormScale", max := "Parameters"."Cab Angle Max deg", out => "Cab Angle Real Meter")
   END_RUNG
   // the same network as SCL:
   #"Cab Angle NormScale" := NORM_X(MIN := "Parameters"."Cab Angle Min", VALUE := "Cabin Angle", MAX := "Parameters"."Cab Angle Max");
   "Cab Angle Real Meter" := SCALE_X(MIN := "Parameters"."Cab Angle Min deg", VALUE := #"Cab Angle NormScale", MAX := "Parameters"."Cab Angle Max deg");
END_REGION

REGION Network 3: Cabin Left Stop Limit
   RUNG wire#powerrail
      I_Contact( "Button ByPass" )
      wire#w1
      { S7_Templates := "SrcType := Real" } LE_Contact(in1 := "Cab Angle Real Meter", in2 := "Parameters"."Cabin Stop Point Left")
      { S7_Templates := "time_type := Time" } "Cab Angle Left Timer".TOF(pt := T#0.5s, et =>)
      Coil( "Cab Angle Left Stop" )
   END_RUNG
   RUNG wire#w1
      I_Contact( "Cabin LSW Left" )
      Contact( "sanal kesici (1)" )
      Coil( "Cab LS Left Stop" )
   END_RUNG
   RUNG wire#powerrail
      Contact( "Cab Angle Left Stop" )
      wire#w2
      Coil( "Cab Stop Left All" )
   END_RUNG
   RUNG wire#powerrail
      Contact( "Cab LS Left Stop" )
   END_RUNG wire#w2
   // the same network as SCL:
   "Cab Angle Left Timer".TOF(IN := NOT "Button ByPass" AND ("Cab Angle Real Meter" <= "Parameters"."Cabin Stop Point Left"),
                           PT := T#0.5s);
   "Cab Angle Left Stop" := "Cab Angle Left Timer".Q;
   "Cab LS Left Stop" := NOT "Button ByPass" AND NOT "Cabin LSW Left" AND "sanal kesici (1)";
   "Cab Stop Left All" := "Cab Angle Left Stop" OR "Cab LS Left Stop";
END_REGION

REGION Network 4: Cabin Right Stop Limit
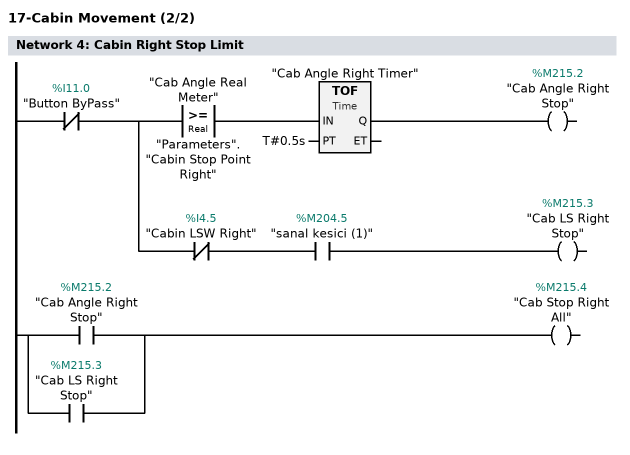
   RUNG wire#powerrail
      I_Contact( "Button ByPass" )
      wire#w1
      { S7_Templates := "SrcType := Real" } GE_Contact(in1 := "Cab Angle Real Meter", in2 := "Parameters"."Cabin Stop Point Right")
      { S7_Templates := "time_type := Time" } "Cab Angle Right Timer".TOF(pt := T#0.5s, et =>)
      Coil( "Cab Angle Right Stop" )
   END_RUNG
   RUNG wire#w1
      I_Contact( "Cabin LSW Right" )
      Contact( "sanal kesici (1)" )
      Coil( "Cab LS Right Stop" )
   END_RUNG
   RUNG wire#powerrail
      Contact( "Cab Angle Right Stop" )
      wire#w2
      Coil( "Cab Stop Right All" )
   END_RUNG
   RUNG wire#powerrail
      Contact( "Cab LS Right Stop" )
   END_RUNG wire#w2
   // the same network as SCL:
   "Cab Angle Right Timer".TOF(IN := NOT "Button ByPass" AND ("Cab Angle Real Meter" >= "Parameters"."Cabin Stop Point Right"),
                           PT := T#0.5s);
   "Cab Angle Right Stop" := "Cab Angle Right Timer".Q;
   "Cab LS Right Stop" := NOT "Button ByPass" AND NOT "Cabin LSW Right" AND "sanal kesici (1)";
   "Cab Stop Right All" := "Cab Angle Right Stop" OR "Cab LS Right Stop";
END_REGION
END_ORGANIZATION_BLOCK

ORGANIZATION_BLOCK "18-Cab Floor"   // OB127, LAD, ProgramCycle
TITLE = "Main Program Sweep (Cycle)"
{ S7_Optimized_Access := 'TRUE' }
VERSION : 0.1
// stored: AutoNumber true, IsIECCheckEnabled false, SetENOAutomatically false
   VAR_INPUT
      Initial_Call : Bool;   // Initial call of this OB
      Remanence : Bool;   // =True, if remanent data are available
   END_VAR
   VAR_TEMP   // added for the SCL form of the ladder/FBD networks
      _w1 : Bool;
   END_VAR
BEGIN

REGION Network 1: Cab Floor Control Manuel & Auto
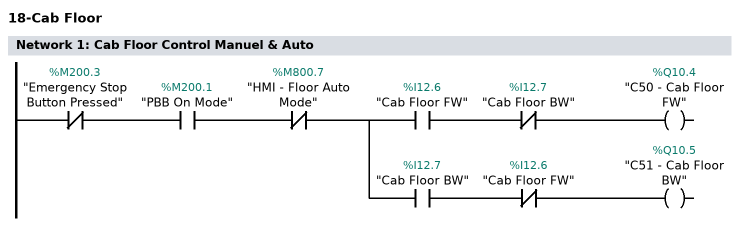
   RUNG wire#powerrail
      I_Contact( "Emergency Stop Button Pressed" )
      Contact( "PBB On Mode" )
      I_Contact( "HMI - Floor Auto Mode" )
      wire#w1
      Contact( "Cab Floor FW" )
      I_Contact( "Cab Floor BW" )
      Coil( "C50 - Cab Floor FW" )
   END_RUNG
   RUNG wire#w1
      Contact( "Cab Floor BW" )
      I_Contact( "Cab Floor FW" )
      Coil( "C51 - Cab Floor BW" )
   END_RUNG
   // the same network as SCL:
   #_w1 := NOT "Emergency Stop Button Pressed" AND "PBB On Mode" AND NOT "HMI - Floor Auto Mode";
   "C50 - Cab Floor FW" := #_w1 AND "Cab Floor FW" AND NOT "Cab Floor BW";
   "C51 - Cab Floor BW" := #_w1 AND "Cab Floor BW" AND NOT "Cab Floor FW";
END_REGION
END_ORGANIZATION_BLOCK

ORGANIZATION_BLOCK "19-Canopy"   // OB129, LAD, ProgramCycle
TITLE = "Main Program Sweep (Cycle)"
{ S7_Optimized_Access := 'TRUE' }
VERSION : 0.1
// stored: AutoNumber true, IsIECCheckEnabled false, SetENOAutomatically false
   VAR_INPUT
      Initial_Call : Bool;   // Initial call of this OB
      Remanence : Bool;   // =True, if remanent data are available
   END_VAR
   VAR_TEMP
      "Temp_1 (NormScale) Wire" : Real;
      "Temp_2 (NormScale) Inclanation" : Real;
      Temp_3 : Real;
      "Temp_4 (Radyan)" : Real;
      Temp_5 : Real;
      "Temp-6 AnimasyonNorm" : Real;
   END_VAR
   VAR_TEMP   // added for the SCL form of the ladder/FBD networks
      _w1 : Bool;
      _w2 : Bool;
      _w3 : Bool;
      _w4 : Bool;
      _w5 : Bool;
      _w6 : Bool;
   END_VAR
BEGIN

REGION Network 1: Canopy
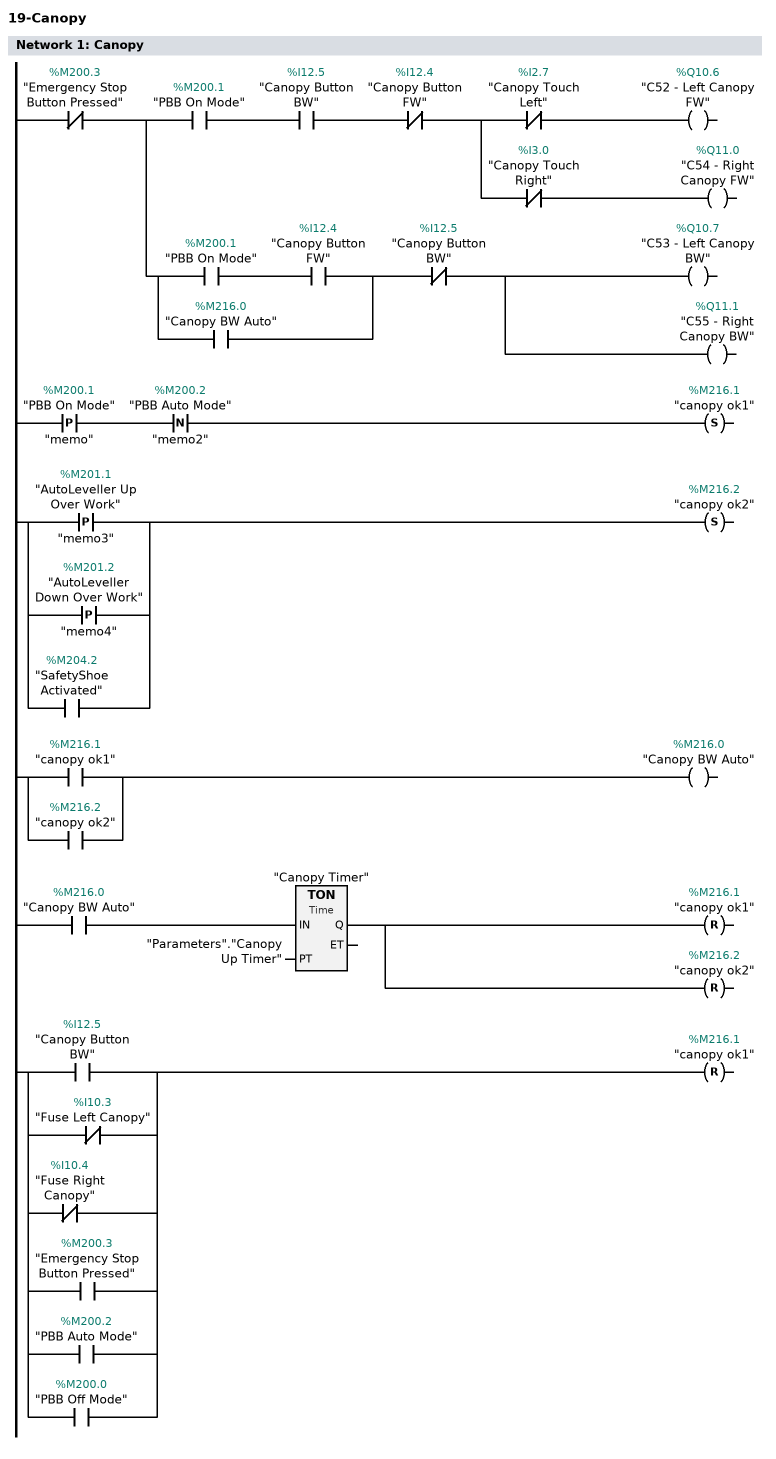
   RUNG wire#powerrail
      I_Contact( "Emergency Stop Button Pressed" )
      wire#w1
      Contact( "PBB On Mode" )
      Contact( "Canopy Button BW" )
      I_Contact( "Canopy Button FW" )
      wire#w2
      I_Contact( "Canopy Touch Left" )
      Coil( "C52 - Left Canopy FW" )
   END_RUNG
   RUNG wire#w2
      I_Contact( "Canopy Touch Right" )
      Coil( "C54 - Right Canopy FW" )
   END_RUNG
   RUNG wire#w1
      Contact( "PBB On Mode" )
      Contact( "Canopy Button FW" )
      wire#w3
      I_Contact( "Canopy Button BW" )
      wire#w4
      Coil( "C53 - Left Canopy BW" )
   END_RUNG
   RUNG wire#w1
      Contact( "Canopy BW Auto" )
   END_RUNG wire#w3
   RUNG wire#w4
      Coil( "C55 - Right Canopy BW" )
   END_RUNG
   RUNG wire#powerrail
      P_Contact(operand := "PBB On Mode", bit := "memo")
      N_Contact(operand := "PBB Auto Mode", bit := "memo2")
      S_Coil( "canopy ok1" )
   END_RUNG
   RUNG wire#powerrail
      P_Contact(operand := "AutoLeveller Up Over Work", bit := "memo3")
      wire#w5
      S_Coil( "canopy ok2" )
   END_RUNG
   RUNG wire#powerrail
      P_Contact(operand := "AutoLeveller Down Over Work", bit := "memo4")
   END_RUNG wire#w5
   RUNG wire#powerrail
      Contact( "SafetyShoe Activated" )
   END_RUNG wire#w5
   RUNG wire#powerrail
      Contact( "canopy ok1" )
      wire#w6
      Coil( "Canopy BW Auto" )
   END_RUNG
   RUNG wire#powerrail
      Contact( "canopy ok2" )
   END_RUNG wire#w6
   RUNG wire#powerrail
      Contact( "Canopy BW Auto" )
      { S7_Templates := "time_type := Time" } "Canopy Timer".TON(pt := "Parameters"."Canopy Up Timer", et =>)
      wire#w7
      R_Coil( "canopy ok1" )
   END_RUNG
   RUNG wire#w7
      R_Coil( "canopy ok2" )
   END_RUNG
   RUNG wire#powerrail
      Contact( "Canopy Button BW" )
      wire#w8
      R_Coil( "canopy ok1" )
   END_RUNG
   RUNG wire#powerrail
      I_Contact( "Fuse Left Canopy" )
   END_RUNG wire#w8
   RUNG wire#powerrail
      I_Contact( "Fuse Right Canopy" )
   END_RUNG wire#w8
   RUNG wire#powerrail
      Contact( "Emergency Stop Button Pressed" )
   END_RUNG wire#w8
   RUNG wire#powerrail
      Contact( "PBB Auto Mode" )
   END_RUNG wire#w8
   RUNG wire#powerrail
      Contact( "PBB Off Mode" )
   END_RUNG wire#w8
   // the same network as SCL:
   #_w1 := NOT "Emergency Stop Button Pressed";
   #_w2 := #_w1 AND "PBB On Mode" AND "Canopy Button BW" AND NOT "Canopy Button FW";
   "C52 - Left Canopy FW" := #_w2 AND NOT "Canopy Touch Left";
   "C54 - Right Canopy FW" := #_w2 AND NOT "Canopy Touch Right";
   "C53 - Left Canopy BW" := #_w1 AND (("PBB On Mode" AND "Canopy Button FW") OR "Canopy BW Auto") AND NOT "Canopy Button BW";
   "C55 - Right Canopy BW" := "C53 - Left Canopy BW";
   #_w3 := "PBB On Mode" AND NOT "memo";   // rising edge of "PBB On Mode"
   "memo" := "PBB On Mode";
   #_w4 := #_w3 AND NOT "PBB Auto Mode" AND "memo2";   // falling edge of "PBB Auto Mode"
   "memo2" := "PBB Auto Mode";
   IF #_w4 THEN "canopy ok1" := TRUE; END_IF;
   #_w5 := "AutoLeveller Up Over Work" AND NOT "memo3";   // rising edge of "AutoLeveller Up Over Work"
   "memo3" := "AutoLeveller Up Over Work";
   #_w6 := "AutoLeveller Down Over Work" AND NOT "memo4";   // rising edge of "AutoLeveller Down Over Work"
   "memo4" := "AutoLeveller Down Over Work";
   IF #_w5 OR #_w6 OR "SafetyShoe Activated" THEN "canopy ok2" := TRUE; END_IF;
   "Canopy BW Auto" := "canopy ok1" OR "canopy ok2";
   "Canopy Timer".TON(IN := "Canopy BW Auto", PT := "Parameters"."Canopy Up Timer");
   IF "Canopy Timer".Q THEN
       "canopy ok1" := FALSE;
       "canopy ok2" := FALSE;
   END_IF;
   IF "Canopy Button BW" OR NOT "Fuse Left Canopy" OR NOT "Fuse Right Canopy" OR "Emergency Stop Button Pressed" OR "PBB Auto Mode" OR "PBB Off Mode" THEN
       "canopy ok1" := FALSE;
   END_IF;
END_REGION
END_ORGANIZATION_BLOCK

ORGANIZATION_BLOCK "20-Autoleveler"   // OB133, LAD, ProgramCycle
TITLE = "Main Program Sweep (Cycle)"
{ S7_Optimized_Access := 'TRUE' }
VERSION : 0.1
// stored: AutoNumber true, IsIECCheckEnabled false, SetENOAutomatically false
   VAR_INPUT
      Initial_Call : Bool;   // Initial call of this OB
      Remanence : Bool;   // =True, if remanent data are available
   END_VAR
   VAR_TEMP   // added for the SCL form of the ladder/FBD networks
      _w1 : Bool;
      _w2 : Bool;
   END_VAR
BEGIN

REGION Network 1: AutoLeveller Definition
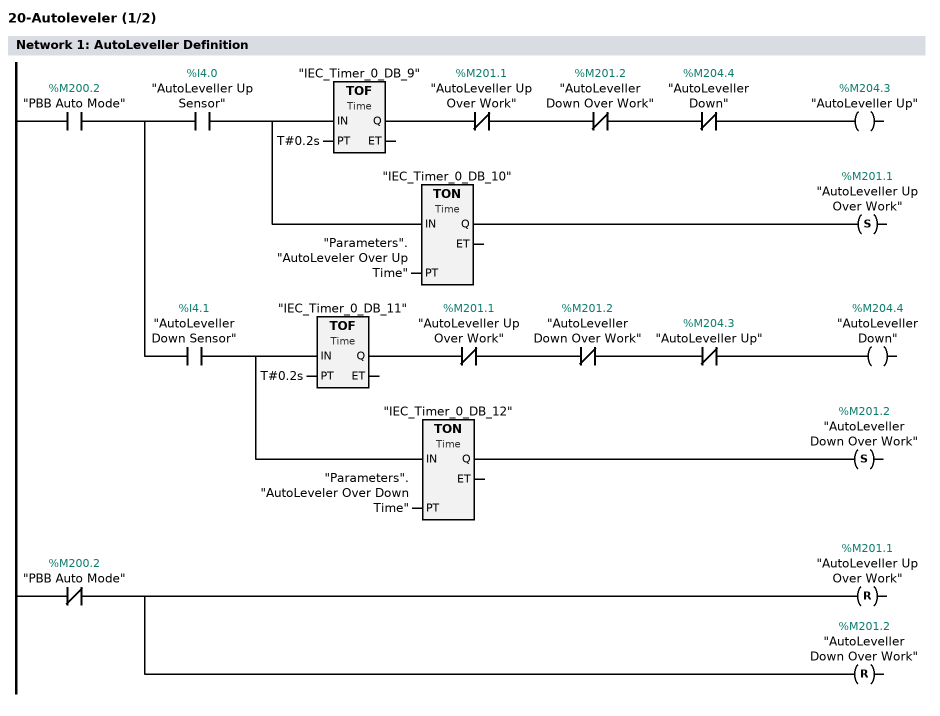
   RUNG wire#powerrail
      Contact( "PBB Auto Mode" )
      wire#w1
      Contact( "AutoLeveller Up Sensor" )
      wire#w2
      { S7_Templates := "time_type := Time" } "IEC_Timer_0_DB_9".TOF(pt := T#0.2s, et =>)
      I_Contact( "AutoLeveller Up Over Work" )
      I_Contact( "AutoLeveller Down Over Work" )
      I_Contact( "AutoLeveller Down" )
      Coil( "AutoLeveller Up" )
   END_RUNG
   RUNG wire#w2
      { S7_Templates := "time_type := Time" } "IEC_Timer_0_DB_10".TON(pt := "Parameters"."AutoLeveler Over Up Time", et =>)
      S_Coil( "AutoLeveller Up Over Work" )
   END_RUNG
   RUNG wire#w1
      Contact( "AutoLeveller Down Sensor" )
      wire#w3
      { S7_Templates := "time_type := Time" } "IEC_Timer_0_DB_11".TOF(pt := T#0.2s, et =>)
      I_Contact( "AutoLeveller Up Over Work" )
      I_Contact( "AutoLeveller Down Over Work" )
      I_Contact( "AutoLeveller Up" )
      Coil( "AutoLeveller Down" )
   END_RUNG
   RUNG wire#w3
      { S7_Templates := "time_type := Time" } "IEC_Timer_0_DB_12".TON(pt := "Parameters"."AutoLeveler Over Down Time", et =>)
      S_Coil( "AutoLeveller Down Over Work" )
   END_RUNG
   RUNG wire#powerrail
      I_Contact( "PBB Auto Mode" )
      wire#w4
      R_Coil( "AutoLeveller Up Over Work" )
   END_RUNG
   RUNG wire#w4
      R_Coil( "AutoLeveller Down Over Work" )
   END_RUNG
   // the same network as SCL:
   #_w1 := "PBB Auto Mode" AND "AutoLeveller Up Sensor";
   "IEC_Timer_0_DB_9".TOF(IN := #_w1, PT := T#0.2s);
   "AutoLeveller Up" := "IEC_Timer_0_DB_9".Q AND NOT "AutoLeveller Up Over Work" AND NOT "AutoLeveller Down Over Work" AND NOT "AutoLeveller Down";
   "IEC_Timer_0_DB_10".TON(IN := #_w1, PT := "Parameters"."AutoLeveler Over Up Time");
   IF "IEC_Timer_0_DB_10".Q THEN "AutoLeveller Up Over Work" := TRUE; END_IF;
   #_w2 := "PBB Auto Mode" AND "AutoLeveller Down Sensor";
   "IEC_Timer_0_DB_11".TOF(IN := #_w2, PT := T#0.2s);
   "AutoLeveller Down" := "IEC_Timer_0_DB_11".Q AND NOT "AutoLeveller Up Over Work" AND NOT "AutoLeveller Down Over Work" AND NOT "AutoLeveller Up";
   "IEC_Timer_0_DB_12".TON(IN := #_w2, PT := "Parameters"."AutoLeveler Over Down Time");
   IF "IEC_Timer_0_DB_12".Q THEN "AutoLeveller Down Over Work" := TRUE; END_IF;
   IF NOT "PBB Auto Mode" THEN
       "AutoLeveller Up Over Work" := FALSE;
       "AutoLeveller Down Over Work" := FALSE;
   END_IF;
END_REGION

REGION Network 2: AutoLeveller Motor
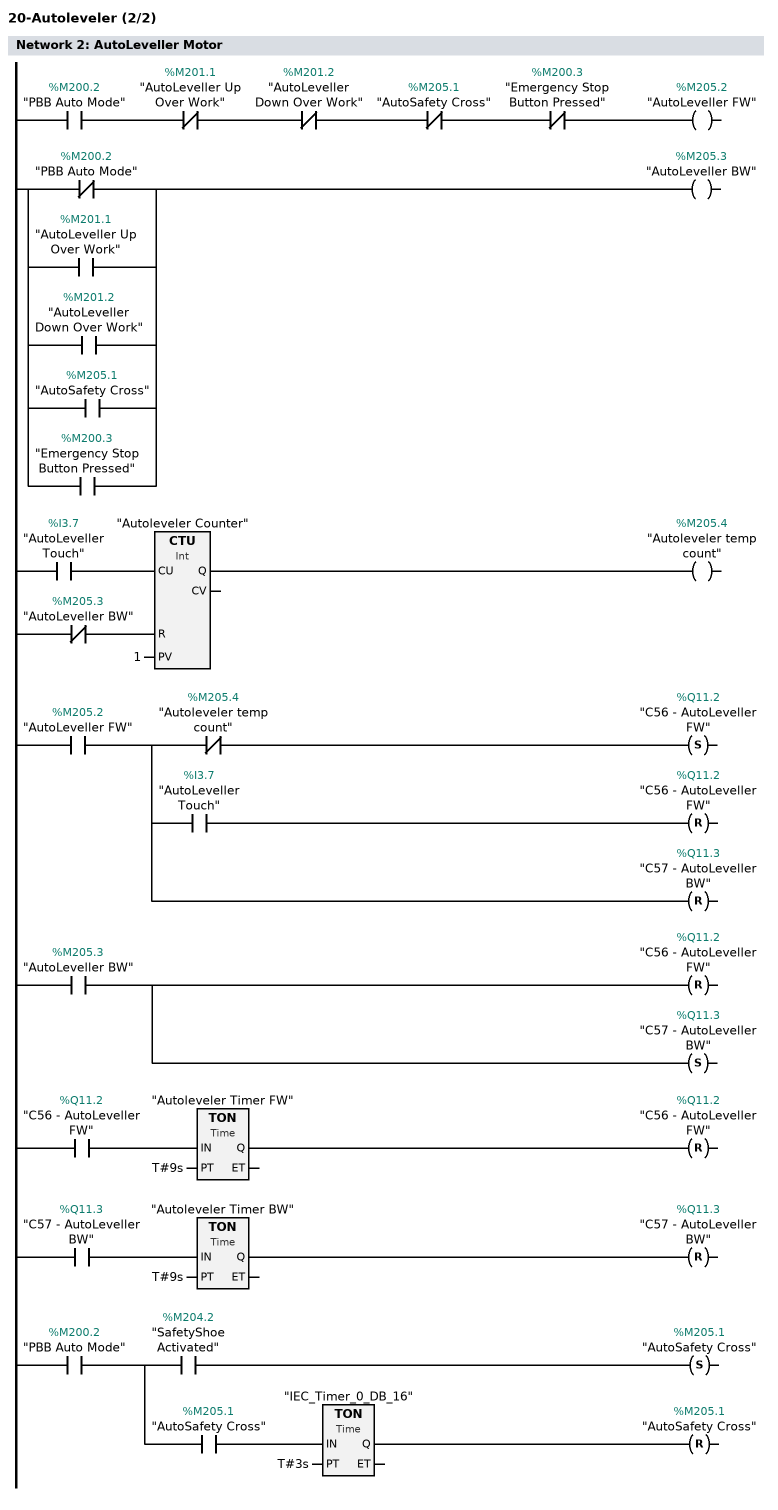
   RUNG wire#powerrail
      Contact( "PBB Auto Mode" )
      I_Contact( "AutoLeveller Up Over Work" )
      I_Contact( "AutoLeveller Down Over Work" )
      I_Contact( "AutoSafety Cross" )
      I_Contact( "Emergency Stop Button Pressed" )
      Coil( "AutoLeveller FW" )
   END_RUNG
   RUNG wire#powerrail
      I_Contact( "PBB Auto Mode" )
      wire#w1
      Coil( "AutoLeveller BW" )
   END_RUNG
   RUNG wire#powerrail
      Contact( "AutoLeveller Up Over Work" )
   END_RUNG wire#w1
   RUNG wire#powerrail
      Contact( "AutoLeveller Down Over Work" )
   END_RUNG wire#w1
   RUNG wire#powerrail
      Contact( "AutoSafety Cross" )
   END_RUNG wire#w1
   RUNG wire#powerrail
      Contact( "Emergency Stop Button Pressed" )
   END_RUNG wire#w1
   RUNG wire#powerrail
      Contact( "AutoLeveller Touch" )
      { S7_Templates := "value_type := Int" } "Autoleveler Counter".CTU(r := wire#w2, pv := 1, cv =>)
      Coil( "Autoleveler temp count" )
   END_RUNG
   RUNG wire#powerrail
      I_Contact( "AutoLeveller BW" )
   END_RUNG wire#w2
   RUNG wire#powerrail
      Contact( "AutoLeveller FW" )
      wire#w3
      I_Contact( "Autoleveler temp count" )
      S_Coil( "C56 - AutoLeveller FW" )
   END_RUNG
   RUNG wire#w3
      Contact( "AutoLeveller Touch" )
      R_Coil( "C56 - AutoLeveller FW" )
   END_RUNG
   RUNG wire#w3
      R_Coil( "C57 - AutoLeveller BW" )
   END_RUNG
   RUNG wire#powerrail
      Contact( "AutoLeveller BW" )
      wire#w4
      R_Coil( "C56 - AutoLeveller FW" )
   END_RUNG
   RUNG wire#w4
      S_Coil( "C57 - AutoLeveller BW" )
   END_RUNG
   RUNG wire#powerrail
      Contact( "C56 - AutoLeveller FW" )
      { S7_Templates := "time_type := Time" } "Autoleveler Timer FW".TON(pt := T#9s, et =>)
      R_Coil( "C56 - AutoLeveller FW" )
   END_RUNG
   RUNG wire#powerrail
      Contact( "C57 - AutoLeveller BW" )
      { S7_Templates := "time_type := Time" } "Autoleveler Timer BW".TON(pt := T#9s, et =>)
      R_Coil( "C57 - AutoLeveller BW" )
   END_RUNG
   RUNG wire#powerrail
      Contact( "PBB Auto Mode" )
      wire#w5
      Contact( "SafetyShoe Activated" )
      S_Coil( "AutoSafety Cross" )
   END_RUNG
   RUNG wire#w5
      Contact( "AutoSafety Cross" )
      { S7_Templates := "time_type := Time" } "IEC_Timer_0_DB_16".TON(pt := T#3s, et =>)
      R_Coil( "AutoSafety Cross" )
   END_RUNG
   // the same network as SCL:
   "AutoLeveller FW" := "PBB Auto Mode" AND NOT "AutoLeveller Up Over Work" AND NOT "AutoLeveller Down Over Work" AND NOT "AutoSafety Cross" AND NOT "Emergency Stop Button Pressed";
   "AutoLeveller BW" := NOT "PBB Auto Mode" OR "AutoLeveller Up Over Work" OR "AutoLeveller Down Over Work" OR "AutoSafety Cross" OR "Emergency Stop Button Pressed";
   "Autoleveler Counter".CTU(CU := "AutoLeveller Touch", R := NOT "AutoLeveller BW", PV := 1);
   "Autoleveler temp count" := "Autoleveler Counter".Q;
   IF "AutoLeveller FW" AND NOT "Autoleveler temp count" THEN "C56 - AutoLeveller FW" := TRUE; END_IF;
   IF "AutoLeveller FW" AND "AutoLeveller Touch" THEN "C56 - AutoLeveller FW" := FALSE; END_IF;
   IF "AutoLeveller FW" THEN "C57 - AutoLeveller BW" := FALSE; END_IF;
   IF "AutoLeveller BW" THEN
       "C56 - AutoLeveller FW" := FALSE;
       "C57 - AutoLeveller BW" := TRUE;
   END_IF;
   "Autoleveler Timer FW".TON(IN := "C56 - AutoLeveller FW", PT := T#9s);
   IF "Autoleveler Timer FW".Q THEN "C56 - AutoLeveller FW" := FALSE; END_IF;
   "Autoleveler Timer BW".TON(IN := "C57 - AutoLeveller BW", PT := T#9s);
   IF "Autoleveler Timer BW".Q THEN "C57 - AutoLeveller BW" := FALSE; END_IF;
   IF "PBB Auto Mode" AND "SafetyShoe Activated" THEN "AutoSafety Cross" := TRUE; END_IF;
   "IEC_Timer_0_DB_16".TON(IN := "PBB Auto Mode" AND "AutoSafety Cross", PT := T#3s);
   IF "IEC_Timer_0_DB_16".Q THEN "AutoSafety Cross" := FALSE; END_IF;
END_REGION
END_ORGANIZATION_BLOCK

ORGANIZATION_BLOCK "21-SafetyShoe"   // OB134, LAD, ProgramCycle
TITLE = "Main Program Sweep (Cycle)"
{ S7_Optimized_Access := 'TRUE' }
VERSION : 0.1
// stored: AutoNumber true, IsIECCheckEnabled false, SetENOAutomatically false
   VAR_INPUT
      Initial_Call : Bool;   // Initial call of this OB
      Remanence : Bool;   // =True, if remanent data are available
   END_VAR
   VAR_TEMP   // added for the SCL form of the ladder/FBD networks
      _w1 : Bool;
   END_VAR
BEGIN

REGION Network 1: SafetyShoe
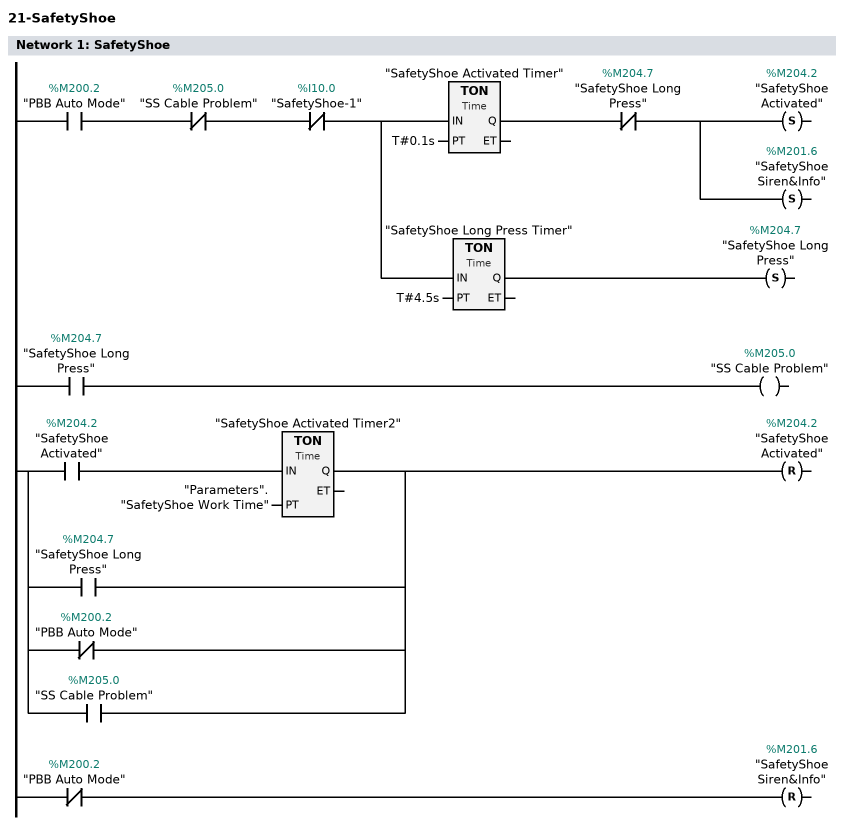
   RUNG wire#powerrail
      Contact( "PBB Auto Mode" )
      I_Contact( "SS Cable Problem" )
      I_Contact( "SafetyShoe-1" )
      wire#w1
      { S7_Templates := "time_type := Time" } "SafetyShoe Activated Timer".TON(pt := T#0.1s, et =>)
      I_Contact( "SafetyShoe Long Press" )
      wire#w2
      S_Coil( "SafetyShoe Activated" )
   END_RUNG
   RUNG wire#w2
      S_Coil( "SafetyShoe Siren&Info" )
   END_RUNG
   RUNG wire#w1
      { S7_Templates := "time_type := Time" } "SafetyShoe Long Press Timer".TON(pt := T#4.5s, et =>)
      S_Coil( "SafetyShoe Long Press" )
   END_RUNG
   RUNG wire#powerrail
      Contact( "SafetyShoe Long Press" )
      Coil( "SS Cable Problem" )
   END_RUNG
   RUNG wire#powerrail
      Contact( "SafetyShoe Activated" )
      { S7_Templates := "time_type := Time" } "SafetyShoe Activated Timer2".TON(pt := "Parameters"."SafetyShoe Work Time", et =>)
      wire#w3
      R_Coil( "SafetyShoe Activated" )
   END_RUNG
   RUNG wire#powerrail
      Contact( "SafetyShoe Long Press" )
   END_RUNG wire#w3
   RUNG wire#powerrail
      I_Contact( "PBB Auto Mode" )
   END_RUNG wire#w3
   RUNG wire#powerrail
      Contact( "SS Cable Problem" )
   END_RUNG wire#w3
   RUNG wire#powerrail
      I_Contact( "PBB Auto Mode" )
      R_Coil( "SafetyShoe Siren&Info" )
   END_RUNG
   // the same network as SCL:
   #_w1 := "PBB Auto Mode" AND NOT "SS Cable Problem" AND NOT "SafetyShoe-1";
   "SafetyShoe Activated Timer".TON(IN := #_w1, PT := T#0.1s);
   IF "SafetyShoe Activated Timer".Q AND NOT "SafetyShoe Long Press" THEN
       "SafetyShoe Activated" := TRUE;
       "SafetyShoe Siren&Info" := TRUE;
   END_IF;
   "SafetyShoe Long Press Timer".TON(IN := #_w1, PT := T#4.5s);
   IF "SafetyShoe Long Press Timer".Q THEN "SafetyShoe Long Press" := TRUE; END_IF;
   "SS Cable Problem" := "SafetyShoe Long Press";
   "SafetyShoe Activated Timer2".TON(IN := "SafetyShoe Activated", PT := "Parameters"."SafetyShoe Work Time");
   IF "SafetyShoe Activated Timer2".Q OR "SafetyShoe Long Press" OR NOT "PBB Auto Mode" OR "SS Cable Problem" THEN
       "SafetyShoe Activated" := FALSE;
   END_IF;
   IF NOT "PBB Auto Mode" THEN "SafetyShoe Siren&Info" := FALSE; END_IF;
END_REGION
END_ORGANIZATION_BLOCK

DATA_BLOCK "AirCraft Touch Timer"   // DB41
{ S7_Optimized_Access := 'TRUE' }
// stored: AutoNumber true, InstanceOfName IEC_TIMER, OfSystemLibElement IEC_TIMER, OfSystemLibVersion 1.0
"IEC_TIMER"
   // VAR
   //    PT : Time;
   //    ET { ExternalWritable := 'False'} : Time;
   //    IN : Bool;
   //    Q { ExternalWritable := 'False'} : Bool;
   // END_VAR
BEGIN
END_DATA_BLOCK

DATA_BLOCK "Autoleveler Counter"   // DB30
{ S7_Optimized_Access := 'TRUE' }
// stored: AutoNumber true, InstanceOfName IEC_COUNTER, OfSystemLibElement IEC_COUNTER, OfSystemLibVersion 1.0
"IEC_COUNTER"
   // VAR RETAIN
   //    CU : Bool;
   //    CD : Bool;
   //    R : Bool;
   //    LD : Bool;
   //    QU : Bool;
   //    QD : Bool;
   //    PV : Int;
   //    CV : Int;
   // END_VAR
BEGIN
END_DATA_BLOCK

DATA_BLOCK "Autoleveler Timer BW"   // DB44
{ S7_Optimized_Access := 'TRUE' }
// stored: AutoNumber true, InstanceOfName IEC_TIMER, OfSystemLibElement IEC_TIMER, OfSystemLibVersion 1.0
"IEC_TIMER"
   // VAR
   //    PT : Time;
   //    ET { ExternalWritable := 'False'} : Time;
   //    IN : Bool;
   //    Q { ExternalWritable := 'False'} : Bool;
   // END_VAR
BEGIN
END_DATA_BLOCK

DATA_BLOCK "Autoleveler Timer FW"   // DB45
{ S7_Optimized_Access := 'TRUE' }
// stored: AutoNumber true, InstanceOfName IEC_TIMER, OfSystemLibElement IEC_TIMER, OfSystemLibVersion 1.0
"IEC_TIMER"
   // VAR
   //    PT : Time;
   //    ET { ExternalWritable := 'False'} : Time;
   //    IN : Bool;
   //    Q { ExternalWritable := 'False'} : Bool;
   // END_VAR
BEGIN
END_DATA_BLOCK

DATA_BLOCK "Brake Off Timer"   // DB29
{ S7_Optimized_Access := 'TRUE' }
// stored: AutoNumber true, InstanceOfName IEC_TIMER, OfSystemLibElement IEC_TIMER, OfSystemLibVersion 1.0
"IEC_TIMER"
   // VAR
   //    PT : Time;
   //    ET { ExternalWritable := 'False'} : Time;
   //    IN : Bool;
   //    Q { ExternalWritable := 'False'} : Bool;
   // END_VAR
BEGIN
END_DATA_BLOCK

DATA_BLOCK "Brakes On Timer"   // DB28
{ S7_Optimized_Access := 'TRUE' }
// stored: AutoNumber true, InstanceOfName IEC_TIMER, OfSystemLibElement IEC_TIMER, OfSystemLibVersion 1.0
"IEC_TIMER"
   // VAR
   //    PT : Time;
   //    ET { ExternalWritable := 'False'} : Time;
   //    IN : Bool;
   //    Q { ExternalWritable := 'False'} : Bool;
   // END_VAR
BEGIN
END_DATA_BLOCK

DATA_BLOCK "CP - Buzzer Blink"   // DB18
{ S7_Optimized_Access := 'TRUE' }
// stored: InstanceOfName IEC_TIMER, OfSystemLibElement IEC_TIMER, OfSystemLibVersion 1.0
"IEC_TIMER"
   // VAR
   //    PT : Time;
   //    ET { ExternalWritable := 'False'} : Time;
   //    IN : Bool;
   //    Q { ExternalWritable := 'False'} : Bool;
   // END_VAR
BEGIN
END_DATA_BLOCK

DATA_BLOCK "CP - Buzzer Reset"   // DB32
{ S7_Optimized_Access := 'TRUE' }
// stored: InstanceOfName IEC_TIMER, OfSystemLibElement IEC_TIMER, OfSystemLibVersion 1.0
"IEC_TIMER"
   // VAR
   //    PT : Time;
   //    ET { ExternalWritable := 'False'} : Time;
   //    IN : Bool;
   //    Q { ExternalWritable := 'False'} : Bool;
   // END_VAR
BEGIN
END_DATA_BLOCK

DATA_BLOCK "CP - Reset Light Blink"   // DB7
{ S7_Optimized_Access := 'TRUE' }
// stored: AutoNumber true, InstanceOfName IEC_TIMER, OfSystemLibElement IEC_TIMER, OfSystemLibVersion 1.0
"IEC_TIMER"
   // VAR
   //    PT : Time;
   //    ET { ExternalWritable := 'False'} : Time;
   //    IN : Bool;
   //    Q { ExternalWritable := 'False'} : Bool;
   // END_VAR
BEGIN
END_DATA_BLOCK

DATA_BLOCK "CP - Reset Light Reset"   // DB10
{ S7_Optimized_Access := 'TRUE' }
// stored: AutoNumber true, InstanceOfName IEC_TIMER, OfSystemLibElement IEC_TIMER, OfSystemLibVersion 1.0
"IEC_TIMER"
   // VAR
   //    PT : Time;
   //    ET { ExternalWritable := 'False'} : Time;
   //    IN : Bool;
   //    Q { ExternalWritable := 'False'} : Bool;
   // END_VAR
BEGIN
END_DATA_BLOCK

DATA_BLOCK "Cab Angle Left Timer"   // DB4
{ S7_Optimized_Access := 'TRUE' }
// stored: AutoNumber true, InstanceOfName IEC_TIMER, OfSystemLibElement IEC_TIMER, OfSystemLibVersion 1.0
"IEC_TIMER"
   // VAR
   //    PT : Time;
   //    ET { ExternalWritable := 'False'} : Time;
   //    IN : Bool;
   //    Q { ExternalWritable := 'False'} : Bool;
   // END_VAR
BEGIN
END_DATA_BLOCK

DATA_BLOCK "Cab Angle Right Timer"   // DB5
{ S7_Optimized_Access := 'TRUE' }
// stored: AutoNumber true, InstanceOfName IEC_TIMER, OfSystemLibElement IEC_TIMER, OfSystemLibVersion 1.0
"IEC_TIMER"
   // VAR
   //    PT : Time;
   //    ET { ExternalWritable := 'False'} : Time;
   //    IN : Bool;
   //    Q { ExternalWritable := 'False'} : Bool;
   // END_VAR
BEGIN
END_DATA_BLOCK

DATA_BLOCK "Canopy Timer"   // DB3
{ S7_Optimized_Access := 'TRUE' }
// stored: AutoNumber true, InstanceOfName IEC_TIMER, OfSystemLibElement IEC_TIMER, OfSystemLibVersion 1.0
"IEC_TIMER"
   // VAR
   //    PT : Time;
   //    ET { ExternalWritable := 'False'} : Time;
   //    IN : Bool;
   //    Q { ExternalWritable := 'False'} : Bool;
   // END_VAR
BEGIN
END_DATA_BLOCK

DATA_BLOCK "Down Stop Timer"   // DB38
{ S7_Optimized_Access := 'TRUE' }
// stored: AutoNumber true, InstanceOfName IEC_TIMER, OfSystemLibElement IEC_TIMER, OfSystemLibVersion 1.0
"IEC_TIMER"
   // VAR
   //    PT : Time;
   //    ET { ExternalWritable := 'False'} : Time;
   //    IN : Bool;
   //    Q { ExternalWritable := 'False'} : Bool;
   // END_VAR
BEGIN
END_DATA_BLOCK

DATA_BLOCK "HMI Work Off Time"   // DB17
{ S7_Optimized_Access := 'TRUE' }
// stored: AutoNumber true, InstanceOfName IEC_TIMER, OfSystemLibElement IEC_TIMER, OfSystemLibVersion 1.0
"IEC_TIMER"
   // VAR
   //    PT : Time;
   //    ET { ExternalWritable := 'False'} : Time;
   //    IN : Bool;
   //    Q { ExternalWritable := 'False'} : Bool;
   // END_VAR
BEGIN
END_DATA_BLOCK

DATA_BLOCK "IEC_Timer_0_DB"   // DB35
{ S7_Optimized_Access := 'TRUE' }
// stored: AutoNumber true, InstanceOfName IEC_TIMER, OfSystemLibElement IEC_TIMER, OfSystemLibVersion 1.0
"IEC_TIMER"
   // VAR
   //    PT : Time;
   //    ET { ExternalWritable := 'False'} : Time;
   //    IN : Bool;
   //    Q { ExternalWritable := 'False'} : Bool;
   // END_VAR
BEGIN
END_DATA_BLOCK

DATA_BLOCK "IEC_Timer_0_DB_10"   // DB12
{ S7_Optimized_Access := 'TRUE' }
// stored: AutoNumber true, InstanceOfName IEC_TIMER, OfSystemLibElement IEC_TIMER, OfSystemLibVersion 1.0
"IEC_TIMER"
   // VAR
   //    PT : Time;
   //    ET { ExternalWritable := 'False'} : Time;
   //    IN : Bool;
   //    Q { ExternalWritable := 'False'} : Bool;
   // END_VAR
BEGIN
END_DATA_BLOCK

DATA_BLOCK "IEC_Timer_0_DB_11"   // DB13
{ S7_Optimized_Access := 'TRUE' }
// stored: AutoNumber true, InstanceOfName IEC_TIMER, OfSystemLibElement IEC_TIMER, OfSystemLibVersion 1.0
"IEC_TIMER"
   // VAR
   //    PT : Time;
   //    ET { ExternalWritable := 'False'} : Time;
   //    IN : Bool;
   //    Q { ExternalWritable := 'False'} : Bool;
   // END_VAR
BEGIN
END_DATA_BLOCK

DATA_BLOCK "IEC_Timer_0_DB_12"   // DB14
{ S7_Optimized_Access := 'TRUE' }
// stored: AutoNumber true, InstanceOfName IEC_TIMER, OfSystemLibElement IEC_TIMER, OfSystemLibVersion 1.0
"IEC_TIMER"
   // VAR
   //    PT : Time;
   //    ET { ExternalWritable := 'False'} : Time;
   //    IN : Bool;
   //    Q { ExternalWritable := 'False'} : Bool;
   // END_VAR
BEGIN
END_DATA_BLOCK

DATA_BLOCK "IEC_Timer_0_DB_16"   // DB19
{ S7_Optimized_Access := 'TRUE' }
// stored: AutoNumber true, InstanceOfName IEC_TIMER, OfSystemLibElement IEC_TIMER, OfSystemLibVersion 1.0
"IEC_TIMER"
   // VAR
   //    PT : Time;
   //    ET { ExternalWritable := 'False'} : Time;
   //    IN : Bool;
   //    Q { ExternalWritable := 'False'} : Bool;
   // END_VAR
BEGIN
END_DATA_BLOCK

DATA_BLOCK "IEC_Timer_0_DB_22"   // DB25
{ S7_Optimized_Access := 'TRUE' }
// stored: AutoNumber true, InstanceOfName IEC_TIMER, OfSystemLibElement IEC_TIMER, OfSystemLibVersion 1.0
"IEC_TIMER"
   // VAR
   //    PT : Time;
   //    ET { ExternalWritable := 'False'} : Time;
   //    IN : Bool;
   //    Q { ExternalWritable := 'False'} : Bool;
   // END_VAR
BEGIN
END_DATA_BLOCK

DATA_BLOCK "IEC_Timer_0_DB_23"   // DB26
{ S7_Optimized_Access := 'TRUE' }
// stored: AutoNumber true, InstanceOfName IEC_TIMER, OfSystemLibElement IEC_TIMER, OfSystemLibVersion 1.0
"IEC_TIMER"
   // VAR
   //    PT : Time;
   //    ET { ExternalWritable := 'False'} : Time;
   //    IN : Bool;
   //    Q { ExternalWritable := 'False'} : Bool;
   // END_VAR
BEGIN
END_DATA_BLOCK

DATA_BLOCK "IEC_Timer_0_DB_24"   // DB27
{ S7_Optimized_Access := 'TRUE' }
// stored: AutoNumber true, InstanceOfName IEC_TIMER, OfSystemLibElement IEC_TIMER, OfSystemLibVersion 1.0
"IEC_TIMER"
   // VAR
   //    PT : Time;
   //    ET { ExternalWritable := 'False'} : Time;
   //    IN : Bool;
   //    Q { ExternalWritable := 'False'} : Bool;
   // END_VAR
BEGIN
END_DATA_BLOCK

DATA_BLOCK "IEC_Timer_0_DB_4"   // DB6
{ S7_Optimized_Access := 'TRUE' }
// stored: AutoNumber true, InstanceOfName IEC_TIMER, OfSystemLibElement IEC_TIMER, OfSystemLibVersion 1.0
"IEC_TIMER"
   // VAR
   //    PT : Time;
   //    ET { ExternalWritable := 'False'} : Time;
   //    IN : Bool;
   //    Q { ExternalWritable := 'False'} : Bool;
   // END_VAR
BEGIN
END_DATA_BLOCK

DATA_BLOCK "IEC_Timer_0_DB_9"   // DB11
{ S7_Optimized_Access := 'TRUE' }
// stored: AutoNumber true, InstanceOfName IEC_TIMER, OfSystemLibElement IEC_TIMER, OfSystemLibVersion 1.0
"IEC_TIMER"
   // VAR
   //    PT : Time;
   //    ET { ExternalWritable := 'False'} : Time;
   //    IN : Bool;
   //    Q { ExternalWritable := 'False'} : Bool;
   // END_VAR
BEGIN
END_DATA_BLOCK

DATA_BLOCK "JoyStick MID Timer"   // DB43
{ S7_Optimized_Access := 'TRUE' }
// stored: AutoNumber true, InstanceOfName IEC_TIMER, OfSystemLibElement IEC_TIMER, OfSystemLibVersion 1.0
"IEC_TIMER"
   // VAR
   //    PT : Time;
   //    ET { ExternalWritable := 'False'} : Time;
   //    IN : Bool;
   //    Q { ExternalWritable := 'False'} : Bool;
   // END_VAR
BEGIN
END_DATA_BLOCK

DATA_BLOCK "Rotunda LFT Stop"   // DB21
{ S7_Optimized_Access := 'TRUE' }
// stored: AutoNumber true, InstanceOfName IEC_TIMER, OfSystemLibElement IEC_TIMER, OfSystemLibVersion 1.0
"IEC_TIMER"
   // VAR
   //    PT : Time;
   //    ET { ExternalWritable := 'False'} : Time;
   //    IN : Bool;
   //    Q { ExternalWritable := 'False'} : Bool;
   // END_VAR
BEGIN
END_DATA_BLOCK

DATA_BLOCK "Rotunda Right Slow"   // DB20
{ S7_Optimized_Access := 'TRUE' }
// stored: AutoNumber true, InstanceOfName IEC_TIMER, OfSystemLibElement IEC_TIMER, OfSystemLibVersion 1.0
"IEC_TIMER"
   // VAR
   //    PT : Time;
   //    ET { ExternalWritable := 'False'} : Time;
   //    IN : Bool;
   //    Q { ExternalWritable := 'False'} : Bool;
   // END_VAR
BEGIN
END_DATA_BLOCK

DATA_BLOCK "Rotunda Right Stop"   // DB16
{ S7_Optimized_Access := 'TRUE' }
// stored: AutoNumber true, InstanceOfName IEC_TIMER, OfSystemLibElement IEC_TIMER, OfSystemLibVersion 1.0
"IEC_TIMER"
   // VAR
   //    PT : Time;
   //    ET { ExternalWritable := 'False'} : Time;
   //    IN : Bool;
   //    Q { ExternalWritable := 'False'} : Bool;
   // END_VAR
BEGIN
END_DATA_BLOCK

DATA_BLOCK "Rotunda Slow LFT"   // DB36
{ S7_Optimized_Access := 'TRUE' }
// stored: AutoNumber true, InstanceOfName IEC_TIMER, OfSystemLibElement IEC_TIMER, OfSystemLibVersion 1.0
"IEC_TIMER"
   // VAR
   //    PT : Time;
   //    ET { ExternalWritable := 'False'} : Time;
   //    IN : Bool;
   //    Q { ExternalWritable := 'False'} : Bool;
   // END_VAR
BEGIN
END_DATA_BLOCK

DATA_BLOCK "SafetyShoe Activated Timer"   // DB31
{ S7_Optimized_Access := 'TRUE' }
// stored: AutoNumber true, InstanceOfName IEC_TIMER, OfSystemLibElement IEC_TIMER, OfSystemLibVersion 1.0
"IEC_TIMER"
   // VAR
   //    PT : Time;
   //    ET { ExternalWritable := 'False'} : Time;
   //    IN : Bool;
   //    Q { ExternalWritable := 'False'} : Bool;
   // END_VAR
BEGIN
END_DATA_BLOCK

DATA_BLOCK "SafetyShoe Activated Timer2"   // DB34
{ S7_Optimized_Access := 'TRUE' }
// stored: AutoNumber true, InstanceOfName IEC_TIMER, OfSystemLibElement IEC_TIMER, OfSystemLibVersion 1.0
"IEC_TIMER"
   // VAR
   //    PT : Time;
   //    ET { ExternalWritable := 'False'} : Time;
   //    IN : Bool;
   //    Q { ExternalWritable := 'False'} : Bool;
   // END_VAR
BEGIN
END_DATA_BLOCK

DATA_BLOCK "SafetyShoe Long Press Timer"   // DB33
{ S7_Optimized_Access := 'TRUE' }
// stored: AutoNumber true, InstanceOfName IEC_TIMER, OfSystemLibElement IEC_TIMER, OfSystemLibVersion 1.0
"IEC_TIMER"
   // VAR
   //    PT : Time;
   //    ET { ExternalWritable := 'False'} : Time;
   //    IN : Bool;
   //    Q { ExternalWritable := 'False'} : Bool;
   // END_VAR
BEGIN
END_DATA_BLOCK

DATA_BLOCK "SafetyShoe Siren&Info Timer"   // DB15
{ S7_Optimized_Access := 'TRUE' }
// stored: AutoNumber true, InstanceOfName IEC_TIMER, OfSystemLibElement IEC_TIMER, OfSystemLibVersion 1.0
"IEC_TIMER"
   // VAR
   //    PT : Time;
   //    ET { ExternalWritable := 'False'} : Time;
   //    IN : Bool;
   //    Q { ExternalWritable := 'False'} : Bool;
   // END_VAR
BEGIN
END_DATA_BLOCK

DATA_BLOCK "Slow Mode Timer"   // DB37
{ S7_Optimized_Access := 'TRUE' }
// stored: AutoNumber true, InstanceOfName IEC_TIMER, OfSystemLibElement IEC_TIMER, OfSystemLibVersion 1.0
"IEC_TIMER"
   // VAR
   //    PT : Time;
   //    ET { ExternalWritable := 'False'} : Time;
   //    IN : Bool;
   //    Q { ExternalWritable := 'False'} : Bool;
   // END_VAR
BEGIN
END_DATA_BLOCK

DATA_BLOCK "Tunnel BW Slow Timer"   // DB23
{ S7_Optimized_Access := 'TRUE' }
// stored: AutoNumber true, InstanceOfName IEC_TIMER, OfSystemLibElement IEC_TIMER, OfSystemLibVersion 1.0
"IEC_TIMER"
   // VAR
   //    PT : Time;
   //    ET { ExternalWritable := 'False'} : Time;
   //    IN : Bool;
   //    Q { ExternalWritable := 'False'} : Bool;
   // END_VAR
BEGIN
END_DATA_BLOCK

DATA_BLOCK "Tunnel BW Stop Timer"   // DB42
{ S7_Optimized_Access := 'TRUE' }
// stored: AutoNumber true, InstanceOfName IEC_TIMER, OfSystemLibElement IEC_TIMER, OfSystemLibVersion 1.0
"IEC_TIMER"
   // VAR
   //    PT : Time;
   //    ET { ExternalWritable := 'False'} : Time;
   //    IN : Bool;
   //    Q { ExternalWritable := 'False'} : Bool;
   // END_VAR
BEGIN
END_DATA_BLOCK

DATA_BLOCK "Tunnel FW Slow Timer"   // DB22
{ S7_Optimized_Access := 'TRUE' }
// stored: AutoNumber true, InstanceOfName IEC_TIMER, OfSystemLibElement IEC_TIMER, OfSystemLibVersion 1.0
"IEC_TIMER"
   // VAR
   //    PT : Time;
   //    ET { ExternalWritable := 'False'} : Time;
   //    IN : Bool;
   //    Q { ExternalWritable := 'False'} : Bool;
   // END_VAR
BEGIN
END_DATA_BLOCK

DATA_BLOCK "Tunnel FW Stop Timer"   // DB24
{ S7_Optimized_Access := 'TRUE' }
// stored: AutoNumber true, InstanceOfName IEC_TIMER, OfSystemLibElement IEC_TIMER, OfSystemLibVersion 1.0
"IEC_TIMER"
   // VAR
   //    PT : Time;
   //    ET { ExternalWritable := 'False'} : Time;
   //    IN : Bool;
   //    Q { ExternalWritable := 'False'} : Bool;
   // END_VAR
BEGIN
END_DATA_BLOCK

DATA_BLOCK "UltraSonic Craft Timer"   // DB9
{ S7_Optimized_Access := 'TRUE' }
// stored: AutoNumber true, InstanceOfName IEC_TIMER, OfSystemLibElement IEC_TIMER, OfSystemLibVersion 1.0
"IEC_TIMER"
   // VAR
   //    PT : Time;
   //    ET { ExternalWritable := 'False'} : Time;
   //    IN : Bool;
   //    Q { ExternalWritable := 'False'} : Bool;
   // END_VAR
BEGIN
END_DATA_BLOCK

DATA_BLOCK "UltraSonic Timer OFF"   // DB8
{ S7_Optimized_Access := 'TRUE' }
// stored: AutoNumber true, InstanceOfName IEC_TIMER, OfSystemLibElement IEC_TIMER, OfSystemLibVersion 1.0
"IEC_TIMER"
   // VAR
   //    PT : Time;
   //    ET { ExternalWritable := 'False'} : Time;
   //    IN : Bool;
   //    Q { ExternalWritable := 'False'} : Bool;
   // END_VAR
BEGIN
END_DATA_BLOCK

DATA_BLOCK "UltraSonic Timer ON"   // DB2
{ S7_Optimized_Access := 'TRUE' }
// stored: AutoNumber true, InstanceOfName IEC_TIMER, OfSystemLibElement IEC_TIMER, OfSystemLibVersion 1.0
"IEC_TIMER"
   // VAR
   //    PT : Time;
   //    ET { ExternalWritable := 'False'} : Time;
   //    IN : Bool;
   //    Q { ExternalWritable := 'False'} : Bool;
   // END_VAR
BEGIN
END_DATA_BLOCK

DATA_BLOCK "Up Stop Timer"   // DB39
{ S7_Optimized_Access := 'TRUE' }
// stored: AutoNumber true, InstanceOfName IEC_TIMER, OfSystemLibElement IEC_TIMER, OfSystemLibVersion 1.0
"IEC_TIMER"
   // VAR
   //    PT : Time;
   //    ET { ExternalWritable := 'False'} : Time;
   //    IN : Bool;
   //    Q { ExternalWritable := 'False'} : Bool;
   // END_VAR
BEGIN
END_DATA_BLOCK
